// ---- POUs/20_AUTO/Mover/VISU_MoverDetail.TcVIS
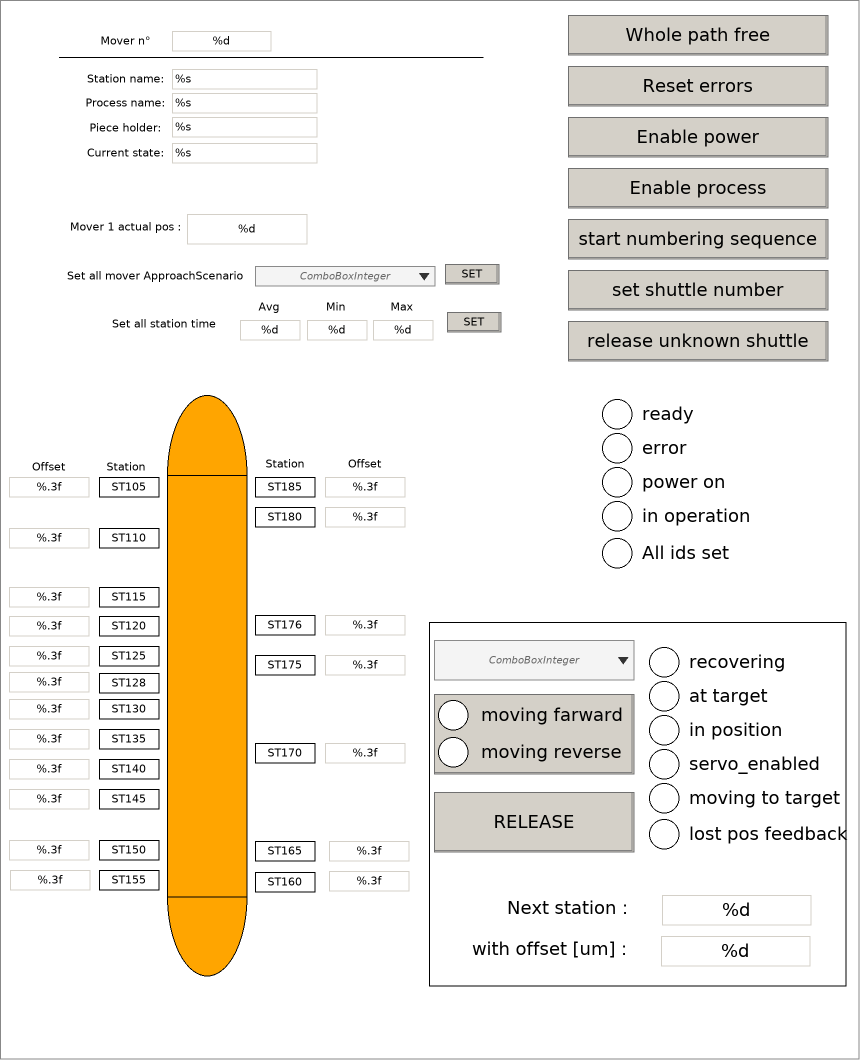
VISUALIZATION VISU_MoverDetail  // 860x1060
    Rectangle (429,622 417x364)
    Button (434,694 200x80)
        toggle gMoverAxis.Q_CT_Shuttle_to_BR.asStruct[HMI.selectedShuttle].bCommand.dirFarward
    Textfield (187,214 120x30), "%d", text variable: MAIN.MoverMan._MoverList[1]._MoverAxis._CurrentPos
        OnMouseDown: write the text variable via Default
    Label (38,212 146x30), "Mover 1 actual pos :"
    ComboBoxInteger (255,266 180x20), variable: MAIN.MoverMan.HMI_Scenario
    Label (59,261 187x30), "Set all mover ApproachScenario"
    Button (445,264 54x20), "SET"
        OnMouseDown: execute { MAIN.MoverMan.SetAllScenario(); }
    Label (93,309 126x30), "Set all station time"
    Textfield (240,320 60x20), "%d", text variable: MAIN.MoverMan.HMI_TimeAvg
        OnMouseDown: write the text variable via Default
    Label (241,296 56x22), "Avg"
    Textfield (307,320 60x20), "%d", text variable: MAIN.MoverMan.HMI_TimeMin
        OnMouseDown: write the text variable via Default
    Label (308,296 56x22), "Min"
    Textfield (373,320 60x20), "%d", text variable: MAIN.MoverMan.HMI_TimeMax
        OnMouseDown: write the text variable via Default
    Label (374,296 56x22), "Max"
    Button (447,312 54x20), "SET"
        OnMouseDown: execute { MAIN.MoverMan.SetAllTimers(ADR(PERS.iStationTimeDef1), 0); MAIN.MoverMan.SetAllTimers(ADR(PERS.iStationTimeDef2), 500); }
    Label (76,26 99x30), "Mover n°"
    Line (59,57) (483,57)
    Label (76,64 99x30), "Station name:"
    Label (76,88 99x30), "Process name:"
    Label (76,113 99x30), "Piece holder:"
    Label (76,138 99x30), "Current state:"
    Textfield (172,31 99x20), "%d", text variable: MAIN.MoverMan.HMI_iSelMover
        OnMouseDown: write the text variable via Default
    Textfield (172,69 145x20), "%s", text variable: MAIN.MoverMan._MoverList[MAIN.MoverMan.HMI_iSelMover].Station.ToString()
    Textfield (172,93 145x20), "%s"
    Textfield (172,117 145x20), "%s", text variable: MAIN.MoverMan._MoverList[MAIN.MoverMan.HMI_iSelMover].AttachedPieceHolder.ToString()
    Textfield (172,143 145x20), "%s", text variable: TO_STRING(MAIN.MoverMan._MoverList[MAIN.MoverMan.HMI_iSelMover]._State)
    Label (79,457 94x20), "Station"
    Label (-1,457 100x20), "Offset"
    Textfield (9,477 80x20), "%.3f", text variable: _20_AUTO.recipe.stationOffsets[StationList_e.ST105]
        OnMouseDown: write the text variable via Default
    Textfield (9,528 80x20), "%.3f", text variable: _20_AUTO.recipe.stationOffsets[StationList_e.ST110]
        OnMouseDown: write the text variable via Default
    Textfield (9,587 80x20), "%.3f", text variable: _20_AUTO.recipe.stationOffsets[StationList_e.ST115]
        OnMouseDown: write the text variable via Default
    Textfield (9,616 80x20), "%.3f", text variable: _20_AUTO.recipe.stationOffsets[StationList_e.ST120]
        OnMouseDown: write the text variable via Default
    Textfield (9,646 80x20), "%.3f", text variable: _20_AUTO.recipe.stationOffsets[StationList_e.ST125]
        OnMouseDown: write the text variable via Default
    Textfield (9,699 80x20), "%.3f", text variable: _20_AUTO.recipe.stationOffsets[StationList_e.ST130]
        OnMouseDown: write the text variable via Default
    Textfield (9,729 80x20), "%.3f", text variable: _20_AUTO.recipe.stationOffsets[StationList_e.ST135]
        OnMouseDown: write the text variable via Default
    Textfield (9,759 80x20), "%.3f", text variable: _20_AUTO.recipe.stationOffsets[StationList_e.ST140]
        OnMouseDown: write the text variable via Default
    Textfield (9,789 80x20), "%.3f", text variable: _20_AUTO.recipe.stationOffsets[StationList_e.ST145]
        OnMouseDown: write the text variable via Default
    Textfield (9,840 80x20), "%.3f", text variable: _20_AUTO.recipe.stationOffsets[StationList_e.ST150]
        OnMouseDown: write the text variable via Default
    Label (315,454 100x20), "Offset"
    Textfield (10,870 80x20), "%.3f", text variable: _20_AUTO.recipe.stationOffsets[StationList_e.ST155]
        OnMouseDown: write the text variable via Default
    Textfield (325,477 80x20), "%.3f", text variable: _20_AUTO.recipe.stationOffsets[StationList_e.ST185]
        OnMouseDown: write the text variable via Default
    Textfield (325,507 80x20), "%.3f", text variable: _20_AUTO.recipe.stationOffsets[StationList_e.ST180]
        OnMouseDown: write the text variable via Default
    Textfield (325,615 80x20), "%.3f", text variable: _20_AUTO.recipe.stationOffsets[StationList_e.ST176]
        OnMouseDown: write the text variable via Default
    Textfield (325,655 80x20), "%.3f", text variable: _20_AUTO.recipe.stationOffsets[StationList_e.ST175]
        OnMouseDown: write the text variable via Default
    Textfield (325,743 80x20), "%.3f", text variable: _20_AUTO.recipe.stationOffsets[StationList_e.ST170]
        OnMouseDown: write the text variable via Default
    Textfield (329,841 80x20), "%.3f", text variable: _20_AUTO.recipe.stationOffsets[StationList_e.ST165]
        OnMouseDown: write the text variable via Default
    Textfield (329,871 80x20), "%.3f", text variable: _20_AUTO.recipe.stationOffsets[StationList_e.ST160]
        OnMouseDown: write the text variable via Default
    Rectangle (99,870 60x20), "ST155", colour toggle: NOT GVL.st155_aut.xMoverPathFree
    Rectangle (99,840 60x20), "ST150", colour toggle: NOT GVL.st150_aut.xMoverPathFree
    Rectangle (99,789 60x20), "ST145", colour toggle: NOT GVL.st145_aut.xMoverPathFree
    Rectangle (99,759 60x20), "ST140", colour toggle: NOT GVL.st140_aut.xMoverPathFree
    Rectangle (99,729 60x20), "ST135", colour toggle: NOT GVL.st135_aut.xMoverPathFree
    Rectangle (99,699 60x20), "ST130", colour toggle: NOT GVL.st130_aut.xMoverPathFree
    Rectangle (99,646 60x20), "ST125", colour toggle: NOT GVL.st125_aut.xMoverPathFree
    Rectangle (99,616 60x20), "ST120", colour toggle: NOT GVL.st120_aut.xMoverPathFree
    Rectangle (99,587 60x20), "ST115", colour toggle: NOT GVL.st115_aut.xMoverPathFree
    Rectangle (99,528 60x20), "ST110", colour toggle: NOT GVL.st110_aut.xMoverPathFree
    Rectangle (99,477 60x20), "ST105", colour toggle: NOT GVL.st105_aut.xMoverPathFree
    Rectangle (255,507 60x20), "ST180", colour toggle: NOT GVL.st180_aut.xMoverPathFree
    Rectangle (255,615 60x20), "ST176", colour toggle: NOT GVL.st176_aut.xMoverPathFree
    Rectangle (255,655 60x20), "ST175", colour toggle: NOT GVL.st175_aut.xMoverPathFree
    Rectangle (255,743 60x20), "ST170", colour toggle: NOT GVL.st170_aut.xMoverPathFree
    Rectangle (255,841 60x20), "ST165", colour toggle: NOT GVL.st165_aut.xMoverPathFree
    Rectangle (255,872 60x20), "ST160", colour toggle: NOT GVL.st160_aut.xMoverPathFree
    Rectangle (255,477 60x20), "ST185", colour toggle: NOT GVL.st185_aut.xMoverPathFree
    Label (238,454 94x20), "Station"
    Ellipse (167,816 80x160)
    Ellipse (167,395 80x160)
    Rectangle (167,475 80x422)
    Button (568,66 260x40), "Reset errors"
        tap gMoverAxis.Q_CT_Track_to_BR.asStruct.bCommand.resetErrors
    Button (568,117 260x40), "Enable power"
        toggle gMoverAxis.Q_CT_Track_to_BR.asStruct.bCommand.enablePower
    ComboBoxInteger (434,640 200x40), variable: HMI.selectedShuttle
    Button (434,792 200x60), "RELEASE", input disabled if: gMoverAxis.Q_CT_Track_to_BR.asStruct.bCommand.enableProcess OR NOT gMoverAxis.I_CT_Track_from_BR.asStruct.bStatus.allIdSet
        tap gMoverAxis.Q_CT_Shuttle_to_BR.asStruct[HMI.selectedShuttle].bCommand.release
    Ellipse (649,647 30x30), colour toggle: gMoverAxis.I_CT_Shuttle_from_BR.asStruct[HMI.selectedShuttle].bStatus.recovering
    Label (686,647 160x30), "recovering"
    Ellipse (649,681 30x30), colour toggle: gMoverAxis.I_CT_Shuttle_from_BR.asStruct[HMI.selectedShuttle].bStatus.at_target
    Label (686,681 160x30), "at target"
    Ellipse (649,715 30x30), colour toggle: gMoverAxis.I_CT_Shuttle_from_BR.asStruct[HMI.selectedShuttle].bStatus.in_position
    Label (686,715 160x30), "in position"
    Ellipse (649,749 30x30), colour toggle: gMoverAxis.I_CT_Shuttle_from_BR.asStruct[HMI.selectedShuttle].bStatus.servo_enabled
    Label (686,749 160x30), "servo_enabled"
    Ellipse (649,783 30x30), colour toggle: gMoverAxis.I_CT_Shuttle_from_BR.asStruct[HMI.selectedShuttle].bStatus.moving_to_load_target
    Label (686,783 160x30), "moving to target"
    Ellipse (649,819 30x30), colour toggle: gMoverAxis.I_CT_Shuttle_from_BR.asStruct[HMI.selectedShuttle].bStatus.lost_position_feedback
    Label (686,819 160x30), "lost pos feedback"
    Ellipse (602,399 30x30), colour toggle: gMoverAxis.I_CT_Track_from_BR.asStruct.bStatus.ready
    Label (639,399 160x30), "ready"
    Ellipse (602,433 30x30), colour toggle: gMoverAxis.I_CT_Track_from_BR.asStruct.bStatus.error
    Label (639,433 160x30), "error"
    Ellipse (602,467 30x30), colour toggle: gMoverAxis.I_CT_Track_from_BR.asStruct.bStatus.powerOn
    Label (639,467 160x30), "power on"
    Ellipse (602,501 30x30), colour toggle: gMoverAxis.I_CT_Track_from_BR.asStruct.bStatus.inOperation
    Label (639,501 160x30), "in operation"
    Button (568,168 260x40), "Enable process"
        toggle gMoverAxis.Q_CT_Track_to_BR.asStruct.bCommand.enableProcess
    Button (568,219 260x40), "start numbering sequence"
        toggle gMoverAxis.Q_CT_Track_to_BR.asStruct.bCommand.startMoverNumberingSequence
    Button (568,270 260x40), "set shuttle number"
        tap gMoverAxis.Q_CT_Track_to_BR.asStruct.bCommand.setShuttleNumber
    Button (568,321 260x40), "release unknown shuttle"
        tap gMoverAxis.Q_CT_Track_to_BR.asStruct.bCommand.releaseUnknownShuttle
    Ellipse (438,700 30x30), colour toggle: gMoverAxis.Q_CT_Shuttle_to_BR.asStruct[HMI.selectedShuttle].bCommand.dirFarward
    Ellipse (438,737 30x30), colour toggle: NOT gMoverAxis.Q_CT_Shuttle_to_BR.asStruct[HMI.selectedShuttle].bCommand.dirFarward
    Label (478,700 160x30), "moving farward"
    Label (478,737 160x30), "moving reverse"
    Button (568,15 260x40), "Whole path free"
        toggle gMoverAxis.Q_CT_Track_to_BR.asStruct.bCommand.wholePathFree
    Textfield (662,895 149x30), "%d", text variable: gMoverAxis.Q_CT_Shuttle_to_BR.asStruct[HMI.selectedShuttle].bNextStation
        OnMouseDown: write the text variable via Default
    Label (471,893 160x30), "Next station :"
    Textfield (661,936 149x30), "%d", text variable: gMoverAxis.Q_CT_Shuttle_to_BR.asStruct[HMI.selectedShuttle].diNextOffset_um
        OnMouseDown: write the text variable via Default
    Label (470,934 160x30), "with offset [um] :"
    Ellipse (602,538 30x30), colour toggle: gMoverAxis.I_CT_Track_from_BR.asStruct.bStatus.allIdSet
    Label (639,538 160x30), "All ids set"
    Textfield (9,672 80x20), "%.3f", text variable: _20_AUTO.recipe.stationOffsets[StationList_e.ST128]
        OnMouseDown: write the text variable via Default
    Rectangle (99,673 60x20), "ST128", colour toggle: NOT GVL.st125_aut.xMoverPathFree
END_VISUALIZATION

// ---- POUs/20_AUTO/Mover/VISU_MoverView.TcVIS
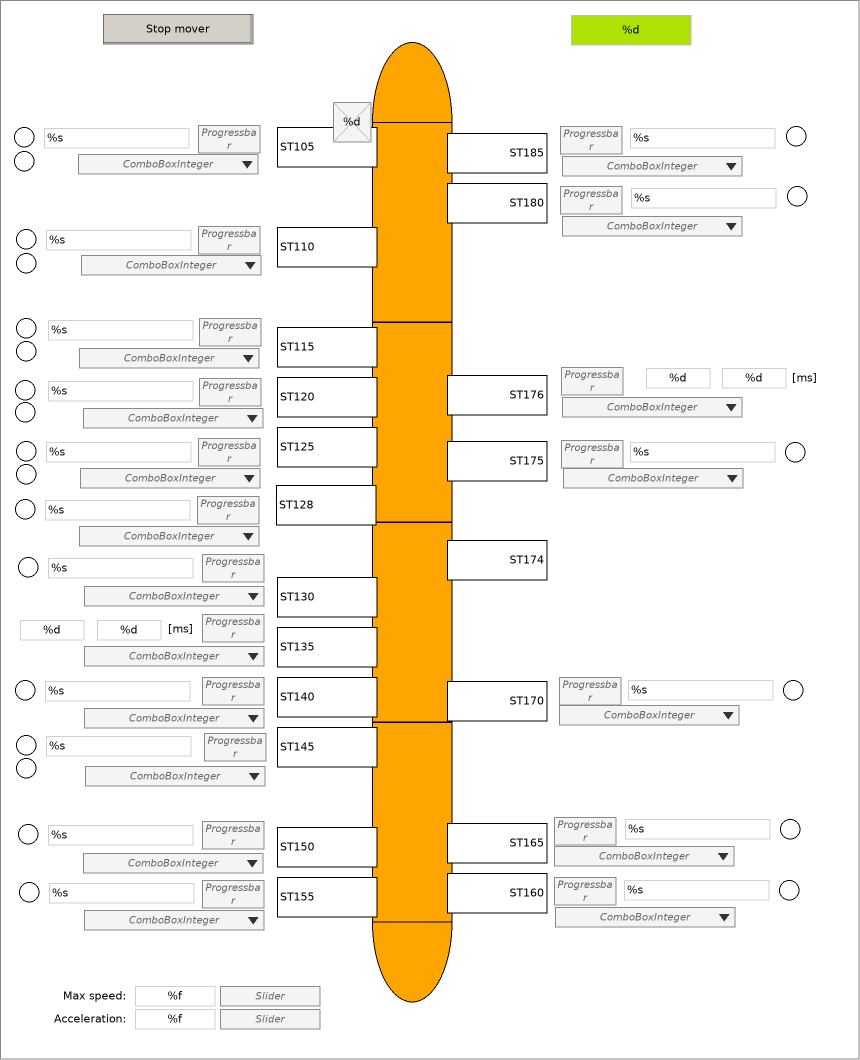
VISUALIZATION VISU_MoverView  // 860x1060
    Ellipse (372,842 80x160)
    Rectangle (372,722 80x200)
    Rectangle (372,522 80x200)
    Rectangle (372,322 80x200)
    Ellipse (372,42 80x160)
    Rectangle (372,122 80x200)
    Rectangle (447,183 100x40), "ST180", colour toggle: NOT GVL.st180_aut.xMoverPathFree
    Rectangle (447,375 100x40), "ST176", colour toggle: NOT GVL.st176_aut.xMoverPathFree
    Rectangle (447,441 100x40), "ST175", colour toggle: NOT GVL.st175_aut.xMoverPathFree
    Rectangle (447,681 100x40), "ST170", colour toggle: NOT GVL.st170_aut.xMoverPathFree
    Rectangle (447,823 100x40), "ST165", colour toggle: NOT GVL.st165_aut.xMoverPathFree
    Rectangle (447,873 100x40), "ST160", colour toggle: NOT GVL.st160_aut.xMoverPathFree
    Rectangle (277,877 100x40), "ST155", colour toggle: NOT GVL.st155_aut.xMoverPathFree
    Rectangle (447,133 100x40), "ST185", colour toggle: NOT GVL.st185_aut.xMoverPathFree
    Progressbar (560,186 62x28), variable: SIMU.iCompletionHMI[18]
    Progressbar (561,367 62x28), variable: SIMU.iCompletionHMI[17]
    Progressbar (561,440 62x28), variable: SIMU.iCompletionHMI[16]
    Progressbar (559,677 62x28), variable: SIMU.iCompletionHMI[14]
    Progressbar (554,817 62x28), variable: SIMU.iCompletionHMI[13]
    Progressbar (554,877 62x28), variable: SIMU.iCompletionHMI[12]
    Progressbar (202,880 62x28), variable: SIMU.iCompletionHMI[11]
    Progressbar (560,126 62x28), variable: SIMU.iCompletionHMI[19]
    Textfield (722,368 64x20), "%d", text variable: PERS.iStationTimeDef2[17]
        OnMouseDown: write the text variable via Default
    Label (777,363 55x30), "[ms]"
    Textfield (571,15 120x30), "%d", text variable: MAIN.MoverMan.PH_num, colour toggle: MAIN.MoverMan.PH_num>2
        OnMouseDown: write the text variable via Default
    ComboBoxInteger (562,156 180x20), variable: MAIN.MoverMan._StationList[18]._ApproachScenario
    ComboBoxInteger (562,216 180x20), variable: MAIN.MoverMan._StationList[17]._ApproachScenario
    ComboBoxInteger (562,397 180x20), variable: MAIN.MoverMan._StationList[16]._ApproachScenario
    ComboBoxInteger (563,468 180x20), variable: MAIN.MoverMan._StationList[16]._ApproachScenario
    ComboBoxInteger (559,705 180x20), variable: MAIN.MoverMan._StationList[14]._ApproachScenario
    ComboBoxInteger (554,846 180x20), variable: MAIN.MoverMan._StationList[13]._ApproachScenario
    ComboBoxInteger (555,907 180x20), variable: MAIN.MoverMan._StationList[12]._ApproachScenario
    ComboBoxInteger (84,910 180x20), variable: MAIN.MoverMan._StationList[11]._ApproachScenario
    Rectangle (277,827 100x40), "ST150", colour toggle: NOT GVL.st150_aut.xMoverPathFree
    Progressbar (202,821 62x28), variable: SIMU.iCompletionHMI[10]
    ComboBoxInteger (83,853 180x20), variable: MAIN.MoverMan._StationList[10]._ApproachScenario
    Rectangle (277,727 100x40), "ST145", colour toggle: NOT GVL.st145_aut.xMoverPathFree
    Progressbar (204,733 62x28), variable: SIMU.iCompletionHMI[9]
    ComboBoxInteger (85,766 180x20), variable: MAIN.MoverMan._StationList[9]._ApproachScenario
    Rectangle (277,677 100x40), "ST140", colour toggle: NOT GVL.st140_aut.xMoverPathFree
    Progressbar (202,677 62x28), variable: SIMU.iCompletionHMI[8]
    ComboBoxInteger (84,708 180x20), variable: MAIN.MoverMan._StationList[8]._ApproachScenario
    Textfield (97,620 64x20), "%d", text variable: PERS.iStationTimeDef2[7]
        OnMouseDown: write the text variable via Default
    Label (153,614 55x30), "[ms]"
    Rectangle (277,627 100x40), "ST135", colour toggle: NOT GVL.st135_aut.xMoverPathFree
    Progressbar (202,614 62x28), variable: SIMU.iCompletionHMI[7]
    ComboBoxInteger (84,646 180x20), variable: MAIN.MoverMan._StationList[7]._ApproachScenario
    Rectangle (277,577 100x40), "ST130", colour toggle: NOT GVL.st130_aut.xMoverPathFree
    Progressbar (202,554 62x28), variable: SIMU.iCompletionHMI[6]
    ComboBoxInteger (84,586 180x20), variable: MAIN.MoverMan._StationList[6]._ApproachScenario
    Rectangle (277,427 100x40), "ST125", colour toggle: NOT GVL.st125_aut.xMoverPathFree
    Progressbar (198,438 62x28), variable: SIMU.iCompletionHMI[5]
    ComboBoxInteger (80,468 180x20), variable: MAIN.MoverMan._StationList[5]._ApproachScenario
    Rectangle (277,377 100x40), "ST120", colour toggle: NOT GVL.st120_aut.xMoverPathFree
    Progressbar (199,378 62x28), variable: SIMU.iCompletionHMI[4]
    ComboBoxInteger (83,408 180x20), variable: MAIN.MoverMan._StationList[4]._ApproachScenario
    Rectangle (277,327 100x40), "ST115", colour toggle: NOT GVL.st115_aut.xMoverPathFree
    Progressbar (199,318 62x28), variable: SIMU.iCompletionHMI[3]
    ComboBoxInteger (79,348 180x20), variable: MAIN.MoverMan._StationList[3]._ApproachScenario
    Rectangle (277,227 100x40), "ST110", colour toggle: NOT GVL.st110_aut.xMoverPathFree
    Progressbar (198,226 62x28), variable: SIMU.iCompletionHMI[2]
    ComboBoxInteger (81,255 180x20), variable: MAIN.MoverMan._StationList[2]._ApproachScenario
    Rectangle (277,127 100x40), "ST105", colour toggle: NOT GVL.st105_aut.xMoverPathFree
    Progressbar (198,125 62x28), variable: SIMU.iCompletionHMI[1]
    ComboBoxInteger (78,154 180x20), variable: MAIN.MoverMan._StationList[1]._ApproachScenario
    Button (103,14 150x30), "Stop mover", colour toggle: MAIN.MoverMan.HMI_xStopMover
        toggle MAIN.MoverMan.HMI_xStopMover
    Textfield (135,986 80x20), "%f", text variable: SIMU.lrSpeedMover
    Textfield (135,1009 80x20), "%f", text variable: SIMU.lrAccelMover
    Label (29,986 100x20), "Max speed:"
    Label (29,1009 100x20), "Acceleration:"
    Slider (220,986 100x20), variable: SIMU.lrSpeedMover, scale 1..50
    Slider (220,1009 100x20), variable: SIMU.lrAccelMoverSlider, scale 0.1..1
    Textfield (20,620 64x20), "%d", text variable: PERS.iStationTimeDef1[7]
        OnMouseDown: write the text variable via Default
    Textfield (646,368 64x20), "%d", text variable: PERS.iStationTimeDef1[17]
        OnMouseDown: write the text variable via Default
    Textfield (46,230 145x20), "%s", text variable: GVL.st110_aut.fb_Pnp.sOUT_Step
    Textfield (48,320 145x20), "%s", text variable: GVL.st115_aut.fb_Pnp.sOUT_Step
    Textfield (48,381 145x20), "%s", text variable: GVL.st120_aut.fb_Pnp.sOUT_Step
    Rectangle (447,540 100x40), "ST174"
    Textfield (46,442 145x20), "%s", text variable: GVL.st125_aut.fb_Pnp.sOUT_Step
    Textfield (46,736 145x20), "%s", text variable: GVL.st145_aut.fb_Pnp.sOUT_Step
    Textfield (631,188 145x20), "%s", text variable: GVL.st180_aut.fb_Pnp.sOUT_Step
    Ellipse (16,229 20x20), colour toggle: GVL.st110_aut.xOUT_Ready
    Ellipse (16,318 20x20), colour toggle: GVL.st115_aut.xOUT_Ready
    Ellipse (15,380 20x20), colour toggle: GVL.st120_aut.xOUT_Ready
    Ellipse (16,441 20x20), colour toggle: GVL.st125_aut.xOUT_Ready
    Ellipse (16,735 20x20), colour toggle: GVL.st145_aut.xOUT_Ready
    Ellipse (787,186 20x20), colour toggle: GVL.st180_aut.xOUT_Ready
    Ellipse (16,253 20x20), colour toggle: GVL.st110_aut.fb_Feeder.xOUT_ErrFlag
    Ellipse (16,341 20x20), colour toggle: GVL.st115_aut.fb_Feeder.xOUT_ErrFlag
    Ellipse (15,402 20x20), colour toggle: GVL.st120_aut.fb_Feeder.xOUT_ErrFlag
    Ellipse (16,464 20x20), colour toggle: GVL.st125_aut.fb_Feeder.xOUT_ErrFlag
    Ellipse (16,758 20x20), colour toggle: GVL.st145_aut.fb_Feeder.xOUT_ErrFlag
    Textfield (630,128 145x20), "%s", text variable: GVL.st185_aut.fb_Pnp.sOUT_Step
    Ellipse (786,126 20x20), colour toggle: GVL.st185_aut.xOUT_Ready
    Textfield (48,558 145x20), "%s", text variable: GVL.st130_aut.fb_Dose.sOUT_Step
    Ellipse (18,557 20x20), colour toggle: GVL.st130_aut.xOUT_Ready
    Textfield (44,128 145x20), "%s", text variable: GVL.st105_aut.fb_Pnp.sOUT_Step
    Ellipse (14,127 20x20), colour toggle: GVL.st105_aut.xOUT_Ready
    Ellipse (14,151 20x20), colour toggle: GVL.st105_aut.fb_Feeder.xOUT_ErrFlag
    Textfield (45,681 145x20), "%s", text variable: GVL.st140_aut.fb_Measure.sOUT_Step
    Ellipse (15,680 20x20), colour toggle: GVL.st140_aut.xOUT_Ready
    Textfield (48,825 145x20), "%s", text variable: GVL.st150_aut.fb_Uss.sOUT_Step
    Ellipse (18,824 20x20), colour toggle: GVL.st150_aut.xOUT_Ready
    Textfield (49,883 145x20), "%s", text variable: GVL.st155_aut.fb_Uss.sOUT_Step
    Ellipse (19,882 20x20), colour toggle: GVL.st155_aut.xOUT_Ready
    Rectangle (276,485 100x40), "ST128", colour toggle: NOT GVL.st128_aut.xMoverPathFree
    Progressbar (197,496 62x28), variable: SIMU.iCompletionHMI[6]
    ComboBoxInteger (79,526 180x20), variable: MAIN.MoverMan._StationList[6]._ApproachScenario
    Textfield (45,500 145x20), "%s", text variable: GVL.st128_aut.fb_TubeCapCheck.sOUT_Step
    Ellipse (15,499 20x20), colour toggle: GVL.st128_aut.xOUT_Ready
    Image (333,102 38x40), "%d", text variable: MAIN.MoverMan._MoverList[1]._ID, colour toggle: MAIN.MoverMan._SimuMoverList[1]._xStuck, invisible if: MAIN.MoverMan._MoverList[1]._MoverAxis._iID>MAIN.MoverMan.MOVER_NUMBER, image: Custom.MoverSimu_final
        p3560616238: MAIN.MoverMan._MoverList[1]._MoverAxis.outSimuCurrentPos.x
        p2738717112: MAIN.MoverMan._MoverList[1]._MoverAxis.outSimuCurrentPos.y
        p2858320360: -MAIN.MoverMan._MoverList[1]._MoverAxis.outSimuCurrentRot
    Image (333,102 38x40), "%d", text variable: MAIN.MoverMan._MoverList[2]._ID, colour toggle: MAIN.MoverMan._SimuMoverList[2]._xStuck, invisible if: MAIN.MoverMan._MoverList[2]._MoverAxis._iID>MAIN.MoverMan.MOVER_NUMBER, image: Custom.MoverSimu_final
        p3560616238: MAIN.MoverMan._MoverList[2]._MoverAxis.outSimuCurrentPos.x
        p2738717112: MAIN.MoverMan._MoverList[2]._MoverAxis.outSimuCurrentPos.y
        p2858320360: -MAIN.MoverMan._MoverList[2]._MoverAxis.outSimuCurrentRot
    Image (333,102 38x40), "%d", text variable: MAIN.MoverMan._MoverList[3]._ID, colour toggle: MAIN.MoverMan._SimuMoverList[3]._xStuck, invisible if: MAIN.MoverMan._MoverList[3]._MoverAxis._iID>MAIN.MoverMan.MOVER_NUMBER, image: Custom.MoverSimu_final
        p3560616238: MAIN.MoverMan._MoverList[3]._MoverAxis.outSimuCurrentPos.x
        p2738717112: MAIN.MoverMan._MoverList[3]._MoverAxis.outSimuCurrentPos.y
        p2858320360: -MAIN.MoverMan._MoverList[3]._MoverAxis.outSimuCurrentRot
    Image (333,102 38x40), "%d", text variable: MAIN.MoverMan._MoverList[4]._ID, colour toggle: MAIN.MoverMan._SimuMoverList[4]._xStuck, invisible if: MAIN.MoverMan._MoverList[4]._MoverAxis._iID>MAIN.MoverMan.MOVER_NUMBER, image: Custom.MoverSimu_final
        p3560616238: MAIN.MoverMan._MoverList[4]._MoverAxis.outSimuCurrentPos.x
        p2738717112: MAIN.MoverMan._MoverList[4]._MoverAxis.outSimuCurrentPos.y
        p2858320360: -MAIN.MoverMan._MoverList[4]._MoverAxis.outSimuCurrentRot
    Image (333,102 38x40), "%d", text variable: MAIN.MoverMan._MoverList[5]._ID, colour toggle: MAIN.MoverMan._SimuMoverList[5]._xStuck, invisible if: MAIN.MoverMan._MoverList[5]._MoverAxis._iID>MAIN.MoverMan.MOVER_NUMBER, image: Custom.MoverSimu_final
        p3560616238: MAIN.MoverMan._MoverList[5]._MoverAxis.outSimuCurrentPos.x
        p2738717112: MAIN.MoverMan._MoverList[5]._MoverAxis.outSimuCurrentPos.y
        p2858320360: -MAIN.MoverMan._MoverList[5]._MoverAxis.outSimuCurrentRot
    Image (333,102 38x40), "%d", text variable: MAIN.MoverMan._MoverList[6]._ID, colour toggle: MAIN.MoverMan._SimuMoverList[6]._xStuck, invisible if: MAIN.MoverMan._MoverList[6]._MoverAxis._iID>MAIN.MoverMan.MOVER_NUMBER, image: Custom.MoverSimu_final
        p3560616238: MAIN.MoverMan._MoverList[6]._MoverAxis.outSimuCurrentPos.x
        p2738717112: MAIN.MoverMan._MoverList[6]._MoverAxis.outSimuCurrentPos.y
        p2858320360: -MAIN.MoverMan._MoverList[6]._MoverAxis.outSimuCurrentRot
    Image (333,102 38x40), "%d", text variable: MAIN.MoverMan._MoverList[7]._ID, colour toggle: MAIN.MoverMan._SimuMoverList[7]._xStuck, invisible if: MAIN.MoverMan._MoverList[7]._MoverAxis._iID>MAIN.MoverMan.MOVER_NUMBER, image: Custom.MoverSimu_final
        p3560616238: MAIN.MoverMan._MoverList[7]._MoverAxis.outSimuCurrentPos.x
        p2738717112: MAIN.MoverMan._MoverList[7]._MoverAxis.outSimuCurrentPos.y
        p2858320360: -MAIN.MoverMan._MoverList[7]._MoverAxis.outSimuCurrentRot
    Image (333,102 38x40), "%d", text variable: MAIN.MoverMan._MoverList[8]._ID, colour toggle: MAIN.MoverMan._SimuMoverList[8]._xStuck, invisible if: MAIN.MoverMan._MoverList[8]._MoverAxis._iID>MAIN.MoverMan.MOVER_NUMBER, image: Custom.MoverSimu_final
        p3560616238: MAIN.MoverMan._MoverList[8]._MoverAxis.outSimuCurrentPos.x
        p2738717112: MAIN.MoverMan._MoverList[8]._MoverAxis.outSimuCurrentPos.y
        p2858320360: -MAIN.MoverMan._MoverList[8]._MoverAxis.outSimuCurrentRot
    Image (333,102 38x40), "%d", text variable: MAIN.MoverMan._MoverList[9]._ID, colour toggle: MAIN.MoverMan._SimuMoverList[9]._xStuck, invisible if: MAIN.MoverMan._MoverList[9]._MoverAxis._iID>MAIN.MoverMan.MOVER_NUMBER, image: Custom.MoverSimu_final
        p3560616238: MAIN.MoverMan._MoverList[9]._MoverAxis.outSimuCurrentPos.x
        p2738717112: MAIN.MoverMan._MoverList[9]._MoverAxis.outSimuCurrentPos.y
        p2858320360: -MAIN.MoverMan._MoverList[9]._MoverAxis.outSimuCurrentRot
    Image (333,102 38x40), "%d", text variable: MAIN.MoverMan._MoverList[10]._ID, colour toggle: MAIN.MoverMan._SimuMoverList[10]._xStuck, invisible if: MAIN.MoverMan._MoverList[10]._MoverAxis._iID>MAIN.MoverMan.MOVER_NUMBER, image: Custom.MoverSimu_final
        p3560616238: MAIN.MoverMan._MoverList[10]._MoverAxis.outSimuCurrentPos.x
        p2738717112: MAIN.MoverMan._MoverList[10]._MoverAxis.outSimuCurrentPos.y
        p2858320360: -MAIN.MoverMan._MoverList[10]._MoverAxis.outSimuCurrentRot
    Image (333,102 38x40), "%d", text variable: MAIN.MoverMan._MoverList[11]._ID, colour toggle: MAIN.MoverMan._SimuMoverList[11]._xStuck, invisible if: MAIN.MoverMan._MoverList[11]._MoverAxis._iID>MAIN.MoverMan.MOVER_NUMBER, image: Custom.MoverSimu_final
        p3560616238: MAIN.MoverMan._MoverList[11]._MoverAxis.outSimuCurrentPos.x
        p2738717112: MAIN.MoverMan._MoverList[11]._MoverAxis.outSimuCurrentPos.y
        p2858320360: -MAIN.MoverMan._MoverList[11]._MoverAxis.outSimuCurrentRot
    Image (333,102 38x40), "%d", text variable: MAIN.MoverMan._MoverList[12]._ID, colour toggle: MAIN.MoverMan._SimuMoverList[12]._xStuck, invisible if: MAIN.MoverMan._MoverList[12]._MoverAxis._iID>MAIN.MoverMan.MOVER_NUMBER, image: Custom.MoverSimu_final
        p3560616238: MAIN.MoverMan._MoverList[12]._MoverAxis.outSimuCurrentPos.x
        p2738717112: MAIN.MoverMan._MoverList[12]._MoverAxis.outSimuCurrentPos.y
        p2858320360: -MAIN.MoverMan._MoverList[12]._MoverAxis.outSimuCurrentRot
    Image (333,102 38x40), "%d", text variable: MAIN.MoverMan._MoverList[13]._ID, colour toggle: MAIN.MoverMan._SimuMoverList[13]._xStuck, invisible if: MAIN.MoverMan._MoverList[13]._MoverAxis._iID>MAIN.MoverMan.MOVER_NUMBER, image: Custom.MoverSimu_final
        p3560616238: MAIN.MoverMan._MoverList[13]._MoverAxis.outSimuCurrentPos.x
        p2738717112: MAIN.MoverMan._MoverList[13]._MoverAxis.outSimuCurrentPos.y
        p2858320360: -MAIN.MoverMan._MoverList[13]._MoverAxis.outSimuCurrentRot
    Image (333,102 38x40), "%d", text variable: MAIN.MoverMan._MoverList[14]._ID, colour toggle: MAIN.MoverMan._SimuMoverList[14]._xStuck, invisible if: MAIN.MoverMan._MoverList[14]._MoverAxis._iID>MAIN.MoverMan.MOVER_NUMBER, image: Custom.MoverSimu_final
        p3560616238: MAIN.MoverMan._MoverList[14]._MoverAxis.outSimuCurrentPos.x
        p2738717112: MAIN.MoverMan._MoverList[14]._MoverAxis.outSimuCurrentPos.y
        p2858320360: -MAIN.MoverMan._MoverList[14]._MoverAxis.outSimuCurrentRot
    Image (333,102 38x40), "%d", text variable: MAIN.MoverMan._MoverList[15]._ID, colour toggle: MAIN.MoverMan._SimuMoverList[15]._xStuck, invisible if: MAIN.MoverMan._MoverList[15]._MoverAxis._iID>MAIN.MoverMan.MOVER_NUMBER, image: Custom.MoverSimu_final
        p3560616238: MAIN.MoverMan._MoverList[15]._MoverAxis.outSimuCurrentPos.x
        p2738717112: MAIN.MoverMan._MoverList[15]._MoverAxis.outSimuCurrentPos.y
        p2858320360: -MAIN.MoverMan._MoverList[15]._MoverAxis.outSimuCurrentRot
    Image (333,102 38x40), "%d", text variable: MAIN.MoverMan._MoverList[16]._ID, colour toggle: MAIN.MoverMan._SimuMoverList[16]._xStuck, invisible if: MAIN.MoverMan._MoverList[16]._MoverAxis._iID>MAIN.MoverMan.MOVER_NUMBER, image: Custom.MoverSimu_final
        p3560616238: MAIN.MoverMan._MoverList[16]._MoverAxis.outSimuCurrentPos.x
        p2738717112: MAIN.MoverMan._MoverList[16]._MoverAxis.outSimuCurrentPos.y
        p2858320360: -MAIN.MoverMan._MoverList[16]._MoverAxis.outSimuCurrentRot
    Image (333,102 38x40), "%d", text variable: MAIN.MoverMan._MoverList[17]._ID, colour toggle: MAIN.MoverMan._SimuMoverList[17]._xStuck, invisible if: MAIN.MoverMan._MoverList[17]._MoverAxis._iID>MAIN.MoverMan.MOVER_NUMBER, image: Custom.MoverSimu_final
        p3560616238: MAIN.MoverMan._MoverList[17]._MoverAxis.outSimuCurrentPos.x
        p2738717112: MAIN.MoverMan._MoverList[17]._MoverAxis.outSimuCurrentPos.y
        p2858320360: -MAIN.MoverMan._MoverList[17]._MoverAxis.outSimuCurrentRot
    Image (333,102 38x40), "%d", text variable: MAIN.MoverMan._MoverList[18]._ID, colour toggle: MAIN.MoverMan._SimuMoverList[18]._xStuck, invisible if: MAIN.MoverMan._MoverList[18]._MoverAxis._iID>MAIN.MoverMan.MOVER_NUMBER, image: Custom.MoverSimu_final
        p3560616238: MAIN.MoverMan._MoverList[18]._MoverAxis.outSimuCurrentPos.x
        p2738717112: MAIN.MoverMan._MoverList[18]._MoverAxis.outSimuCurrentPos.y
        p2858320360: -MAIN.MoverMan._MoverList[18]._MoverAxis.outSimuCurrentRot
    Image (333,102 38x40), "%d", text variable: MAIN.MoverMan._MoverList[19]._ID, colour toggle: MAIN.MoverMan._SimuMoverList[19]._xStuck, invisible if: MAIN.MoverMan._MoverList[19]._MoverAxis._iID>MAIN.MoverMan.MOVER_NUMBER, image: Custom.MoverSimu_final
        p3560616238: MAIN.MoverMan._MoverList[19]._MoverAxis.outSimuCurrentPos.x
        p2738717112: MAIN.MoverMan._MoverList[19]._MoverAxis.outSimuCurrentPos.y
        p2858320360: -MAIN.MoverMan._MoverList[19]._MoverAxis.outSimuCurrentRot
    Textfield (624,880 145x20), "%s", text variable: GVL.st160_aut.fb_ABL_CETA.sOUT_Step
    Ellipse (779,880 20x20), colour toggle: GVL.st160_aut.xOUT_Ready
    Textfield (625,819 145x20), "%s", text variable: GVL.st165_aut.fb_ABL_CETA.sOUT_Step
    Ellipse (780,819 20x20), colour toggle: GVL.st160_aut.xOUT_Ready
    Textfield (628,680 145x20), "%s", text variable: GVL.st170_aut.fb_ABL_RFID.sOUT_Step
    Ellipse (783,680 20x20), colour toggle: GVL.st170_aut.xOUT_Ready
    Textfield (630,442 145x20), "%s", text variable: GVL.st175_aut.fb_laser.sOUT_Step
    Ellipse (785,442 20x20), colour toggle: GVL.st175_aut.xOUT_Ready
END_VISUALIZATION

// ---- POUs/20_AUTO/ST105/VISU_Recipe_ST105.TcVIS
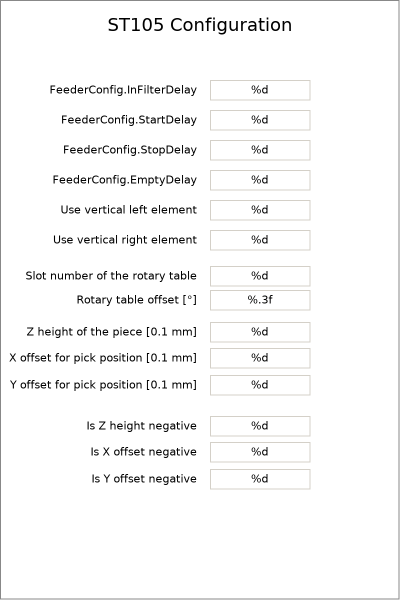
VISUALIZATION VISU_Recipe_ST105  // 400x600
    Textfield (210,80 100x20), "%d", text variable: _20_AUTO.recipe.st110.FeederConfig.InFilterDelay
        OnMouseDown: write the text variable via Default
    Label (0,5 400x40), "ST105 Configuration"
    Label (0,80 200x20), "FeederConfig.InFilterDelay"
    Textfield (210,110 100x20), "%d", text variable: _20_AUTO.recipe.st110.FeederConfig.StartDelay
        OnMouseDown: write the text variable via Default
    Label (0,110 200x20), "FeederConfig.StartDelay"
    Textfield (210,140 100x20), "%d", text variable: _20_AUTO.recipe.st105.FeederConfig.StopDelay
        OnMouseDown: write the text variable via Default
    Label (0,140 200x20), "FeederConfig.StopDelay"
    Textfield (210,170 100x20), "%d", text variable: _20_AUTO.recipe.st105.FeederConfig.EmptyDelay
        OnMouseDown: write the text variable via Default
    Label (0,170 200x20), "FeederConfig.EmptyDelay"
    Label (0,200 200x20), "Use vertical left element"
    Label (0,230 200x20), "Use vertical right element"
    Textfield (210,200 100x20), "%d", text variable: _20_AUTO.recipe.st105.xUseVerLeft
        OnMouseDown: write the text variable via Default
    Textfield (210,230 100x20), "%d", text variable: _20_AUTO.recipe.st105.xUseVerRight
        OnMouseDown: write the text variable via Default
    Textfield (210,416 100x20), "%d", text variable: _20_AUTO.recipe.st105.isPickUpPos_Z_neg
        OnMouseDown: write the text variable via Default
    Label (0,442 200x20), "Is X offset negative"
    Textfield (210,442 100x20), "%d", text variable: _20_AUTO.recipe.st105.isPickOffset_X_neg
        OnMouseDown: write the text variable via Default
    Label (0,469 200x20), "Is Y offset negative"
    Textfield (210,469 100x20), "%d", text variable: _20_AUTO.recipe.st105.isPickOffset_Y_neg
        OnMouseDown: write the text variable via Default
    Label (0,416 200x20), "Is Z height negative"
    Textfield (210,322 100x20), "%d", text variable: _20_AUTO.recipe.st105.PickUpPos_Z_deci
        OnMouseDown: write the text variable via Default
    Label (0,348 200x20), "X offset for pick position [0.1 mm]"
    Textfield (210,348 100x20), "%d", text variable: _20_AUTO.recipe.st105.PickOffset_X_deci
        OnMouseDown: write the text variable via Default
    Label (0,375 200x20), "Y offset for pick position [0.1 mm]"
    Textfield (210,375 100x20), "%d", text variable: _20_AUTO.recipe.st105.PickOffset_Y_deci
        OnMouseDown: write the text variable via Default
    Label (0,322 200x20), "Z height of the piece [0.1 mm]"
    Label (0,266 200x20), "Slot number of the rotary table"
    Textfield (210,266 100x20), "%d", text variable: _20_AUTO.recipe.st105.FeederSize
        OnMouseDown: write the text variable via Default
    Textfield (210,290 100x20), "%.3f", text variable: _20_AUTO.recipe.st105.RotaryTableOffset
        OnMouseDown: write the text variable via Default
    Label (0,290 200x20), "Rotary table offset [°]"
END_VISUALIZATION

// ---- POUs/20_AUTO/ST105/VISU_ST105.TcVIS
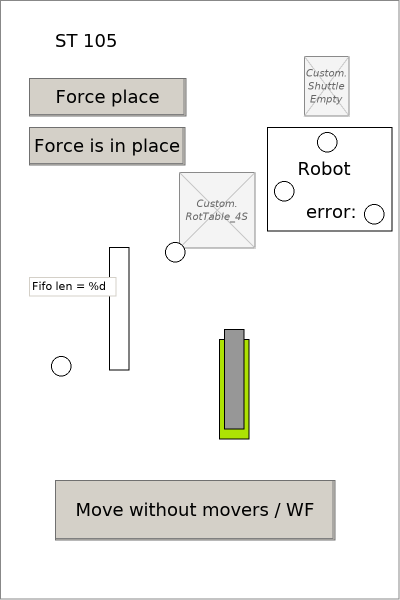
VISUALIZATION VISU_ST105  // 400x600
    Image (304,56 45x60), angle 90, invisible if: NOT __ISVALIDREF(GVL.st105_aut._Mover), image: Custom.Shuttle Empty
    Image (179,172 76x76), angle 45, image: Custom.RotTable_4S
        p2858320360: ST105_Axis.axis105_10W.rActPos
    Rectangle (109,247 20x123), angle 45
    Ellipse (51,356 20x20), colour toggle: GVL.st105_aut.fb_Feeder.simu_feeder.xOUT_NewPiece
    Ellipse (165,242 20x20), colour toggle: GVL.st105_aut.fb_Feeder.simu_feeder.xOUT_NewPiece
    Textfield (29,277 87x19), "Fifo len = %d", text variable: GVL.st105_aut.fb_Feeder.simu_fifo_feeder_to_rotTable.GetLen()
    Label (44,31 85x20), "ST 105"
    Rectangle (219,339 30x100)
    Rectangle (224,329 20x100)
        p2738717112: -GVL.st105_aut.fb_Pnp.fb_simu_axis105_11Z.rOUT_PixActual
    Button (55,480 280x60), "Move without movers / WF", colour toggle: HMI.bArForceCyclusState[StationList_e.ST105]
        tap HMI.btArForceCyclus[StationList_e.ST105].button
    Rectangle (267,127 125x104)
    Ellipse (274,181 20x20), colour toggle: GVL.st105_aut.fb_Pnp.aut_status_from_robot.Picked
    Ellipse (317,132 20x20), colour toggle: GVL.st105_aut.fb_Pnp.aut_status_from_robot.Placed
    Ellipse (364,204 20x20), colour toggle: GVL.st105_aut.fb_Pnp.fanuc_status.Fault
    Label (283,154 82x30), "Robot"
    Label (299,197 65x30), "error:"
    Button (29,78 157x38), "Force place", colour toggle: HMI.bArForceCyclusState[StationList_e.ST105]
        tap GVL.st105_aut.fb_Pnp.hmi_force_place
    Button (29,127 156x38), "Force is in place", colour toggle: HMI.bArForceCyclusState[StationList_e.ST105]
        tap GVL.st105_aut.fb_Pnp.hmi_force_in_place
END_VISUALIZATION

// ---- POUs/20_AUTO/ST110/VISU_Recipe_ST110.TcVIS
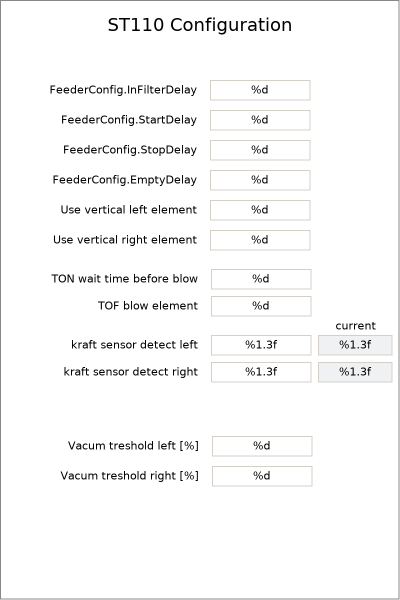
VISUALIZATION VISU_Recipe_ST110  // 400x600
    Textfield (210,80 100x20), "%d", text variable: _20_AUTO.recipe.st110.FeederConfig.InFilterDelay
        OnMouseDown: write the text variable via Default
    Label (0,5 400x40), "ST110 Configuration"
    Label (0,80 200x20), "FeederConfig.InFilterDelay"
    Textfield (210,110 100x20), "%d", text variable: _20_AUTO.recipe.st110.FeederConfig.StartDelay
        OnMouseDown: write the text variable via Default
    Label (0,110 200x20), "FeederConfig.StartDelay"
    Textfield (210,140 100x20), "%d", text variable: _20_AUTO.recipe.st110.FeederConfig.StopDelay
        OnMouseDown: write the text variable via Default
    Label (0,140 200x20), "FeederConfig.StopDelay"
    Textfield (210,170 100x20), "%d", text variable: _20_AUTO.recipe.st110.FeederConfig.EmptyDelay
        OnMouseDown: write the text variable via Default
    Label (0,170 200x20), "FeederConfig.EmptyDelay"
    Label (0,200 200x20), "Use vertical left element"
    Label (0,230 200x20), "Use vertical right element"
    Textfield (210,200 100x20), "%d", text variable: _20_AUTO.recipe.st110.xUseVerLeft
        OnMouseDown: write the text variable via Default
    Textfield (210,230 100x20), "%d", text variable: _20_AUTO.recipe.st110.xUseVerRight
        OnMouseDown: write the text variable via Default
    Label (1,296 200x20), "TOF blow element"
    Textfield (211,296 100x20), "%d", text variable: _20_AUTO.recipe.st110.blowPieceTof_ms
        OnMouseDown: write the text variable via Default
    Label (2,436 200x20), "Vacum treshold left [%]"
    Label (2,466 200x20), "Vacum treshold right [%]"
    Textfield (212,436 100x20), "%d", text variable: _20_AUTO.recipe.st110.vakum_left_pc
        OnMouseDown: write the text variable via Default
    Textfield (212,466 100x20), "%d", text variable: _20_AUTO.recipe.st110.vakum_right_pc
        OnMouseDown: write the text variable via Default
    Label (1,269 200x20), "TON wait time before blow"
    Textfield (211,269 100x20), "%d", text variable: _20_AUTO.recipe.st110.waitBlowPieceTon_ms
        OnMouseDown: write the text variable via Default
    Label (1,362 200x20), "kraft sensor detect right"
    Textfield (211,362 100x20), "%1.3f", text variable: _20_AUTO.recipe.st110.kraft_right_raw
        OnMouseDown: write the text variable via Default
    Label (1,335 200x20), "kraft sensor detect left"
    Textfield (211,335 100x20), "%1.3f", text variable: _20_AUTO.recipe.st110.kraft_left_raw
        OnMouseDown: write the text variable via Default
    Textfield (318,335 74x20), "%1.3f", text variable: GVL.st110_aut.fb_Pnp.fb_kraftLeft.lrOUT_value
        OnMouseDown: write the text variable via Default
    Textfield (318,362 74x20), "%1.3f", text variable: GVL.st110_aut.fb_Pnp.fb_kraftRight.lrOUT_value
        OnMouseDown: write the text variable via Default
    Label (321,316 70x20), "current"
END_VISUALIZATION

// ---- POUs/20_AUTO/ST110/VISU_ST110.TcVIS
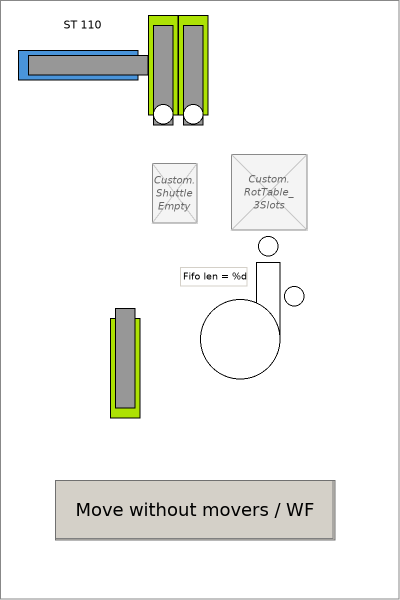
VISUALIZATION VISU_ST110  // 400x600
    Image (152,163 45x60), invisible if: NOT __ISVALIDREF(GVL.st110_aut._Mover), image: Custom.Shuttle Empty
    Image (231,154 76x76), image: Custom.RotTable_3Slots
        p2858320360: ST110_Axis.axis110_10W.rActPos
    Rectangle (18,50 120x30)
    Rectangle (28,55 120x20)
        p3560616238: GVL.st110_aut.fb_Pnp.fb_simu_axis110_01Y.rOUT_PixActual
    Rectangle (148,15 30x100)
        p3560616238: GVL.st110_aut.fb_Pnp.fb_simu_axis110_01Y.rOUT_PixActual
    Rectangle (153,25 20x100)
        p2738717112: GVL.st110_aut.fb_Pnp.fb_simu_axis110_02Z.rOUT_PixActual
        p3560616238: GVL.st110_aut.fb_Pnp.fb_simu_axis110_01Y.rOUT_PixActual
    Rectangle (178,15 30x100)
        p3560616238: GVL.st110_aut.fb_Pnp.fb_simu_axis110_01Y.rOUT_PixActual
    Rectangle (183,25 20x100)
        p2738717112: GVL.st110_aut.fb_Pnp.fb_simu_axis110_03Z.rOUT_PixActual
        p3560616238: GVL.st110_aut.fb_Pnp.fb_simu_axis110_01Y.rOUT_PixActual
    Rectangle (256,262 24x73)
    Ellipse (200,299 80x80), colour toggle: GVL.st110_aut.fb_Feeder.simu_feeder.xIN_Enable
    Ellipse (284,286 20x20), colour toggle: GVL.st110_aut.fb_Feeder.simu_feeder.xOUT_NewPiece
    Ellipse (153,104 20x20), colour toggle: GVL.st110_aut.fb_Pnp.fb_gripperLeft.xIN_AS
        p3560616238: GVL.st110_aut.fb_Pnp.fb_simu_axis110_01Y.rOUT_PixActual
        p2738717112: GVL.st110_aut.fb_Pnp.fb_simu_axis110_02Z.rOUT_PixActual
    Ellipse (183,104 20x20), colour toggle: GVL.st110_aut.fb_Pnp.fb_gripperRight.xIN_AS
        p2738717112: GVL.st110_aut.fb_Pnp.fb_simu_axis110_03Z.rOUT_PixActual
        p3560616238: GVL.st110_aut.fb_Pnp.fb_simu_axis110_01Y.rOUT_PixActual
    Ellipse (258,236 20x20), colour toggle: GVL.st110_aut.fb_Feeder.simu_feeder.xOUT_NewPiece
    Textfield (180,267 67x19), "Fifo len = %d", text variable: GVL.st110_aut.fb_Feeder.simu_fifo_feeder_to_rotTable.GetLen()
    Label (40,15 85x20), "ST 110"
    Rectangle (110,318 30x100)
    Rectangle (115,308 20x100)
        p2738717112: -GVL.st110_aut.fb_Pnp.fb_simu_axis110_04Z.rOUT_PixActual
    Button (55,480 280x60), "Move without movers / WF", colour toggle: HMI.bArForceCyclusState[StationList_e.ST110]
        tap HMI.btArForceCyclus[StationList_e.ST110].button
END_VISUALIZATION

// ---- POUs/20_AUTO/ST115/VISU_Recipe_ST115.TcVIS
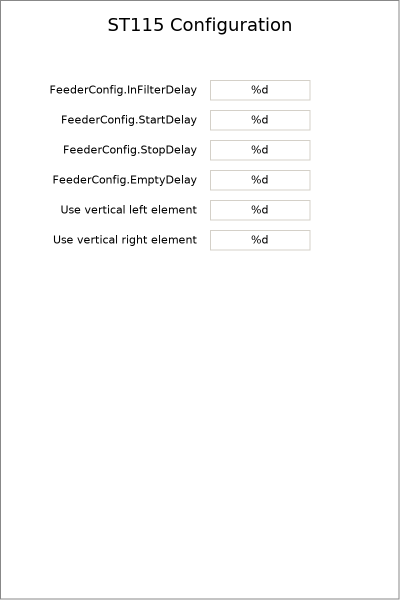
VISUALIZATION VISU_Recipe_ST115  // 400x600
    Textfield (210,80 100x20), "%d", text variable: _20_AUTO.recipe.st115.FeederConfig.InFilterDelay
        OnMouseDown: write the text variable via Default
    Label (0,5 400x40), "ST115 Configuration"
    Label (0,80 200x20), "FeederConfig.InFilterDelay"
    Textfield (210,110 100x20), "%d", text variable: _20_AUTO.recipe.st115.FeederConfig.StartDelay
        OnMouseDown: write the text variable via Default
    Label (0,110 200x20), "FeederConfig.StartDelay"
    Textfield (210,140 100x20), "%d", text variable: _20_AUTO.recipe.st115.FeederConfig.StopDelay
        OnMouseDown: write the text variable via Default
    Label (0,140 200x20), "FeederConfig.StopDelay"
    Textfield (210,170 100x20), "%d", text variable: _20_AUTO.recipe.st115.FeederConfig.EmptyDelay
        OnMouseDown: write the text variable via Default
    Label (0,170 200x20), "FeederConfig.EmptyDelay"
    Label (0,200 200x20), "Use vertical left element"
    Label (0,230 200x20), "Use vertical right element"
    Textfield (210,200 100x20), "%d", text variable: _20_AUTO.recipe.st115.xUseVerLeft
        OnMouseDown: write the text variable via Default
    Textfield (210,230 100x20), "%d", text variable: _20_AUTO.recipe.st115.xUseVerRight
        OnMouseDown: write the text variable via Default
END_VISUALIZATION

// ---- POUs/20_AUTO/ST115/VISU_ST115.TcVIS
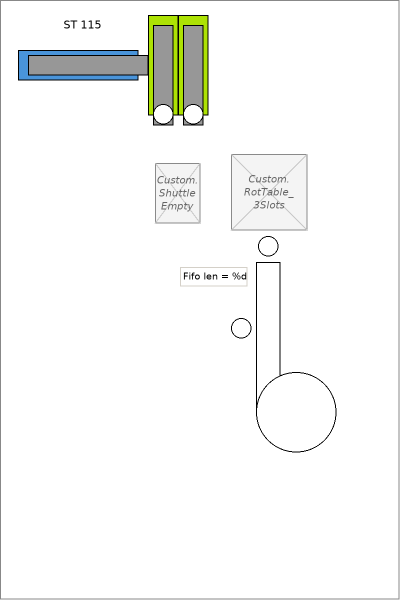
VISUALIZATION VISU_ST115  // 400x600
    Image (155,163 45x60), invisible if: NOT __ISVALIDREF(GVL.st115_aut._Mover), image: Custom.Shuttle Empty
    Image (231,154 76x76), image: Custom.RotTable_3Slots
        p2858320360: ST115_Axis.axis115_10W.rActPos
    Rectangle (18,50 120x30)
    Rectangle (28,55 120x20)
        p3560616238: GVL.st115_aut.fb_Pnp.fb_simu_axis115_01Y.rOUT_PixActual
    Rectangle (148,15 30x100)
        p3560616238: GVL.st115_aut.fb_Pnp.fb_simu_axis115_01Y.rOUT_PixActual
    Rectangle (153,25 20x100)
        p2738717112: GVL.st115_aut.fb_Pnp.fb_simu_axis115_02Z.rOUT_PixActual
        p3560616238: GVL.st115_aut.fb_Pnp.fb_simu_axis115_01Y.rOUT_PixActual
    Rectangle (178,15 30x100)
        p3560616238: GVL.st115_aut.fb_Pnp.fb_simu_axis115_01Y.rOUT_PixActual
    Rectangle (183,25 20x100)
        p2738717112: GVL.st115_aut.fb_Pnp.fb_simu_axis115_03Z.rOUT_PixActual
        p3560616238: GVL.st115_aut.fb_Pnp.fb_simu_axis115_01Y.rOUT_PixActual
    Rectangle (256,262 24x150)
    Ellipse (256,372 80x80), colour toggle: GVL.st115_aut.fb_Feeder.simu_feeder.xIN_Enable
    Ellipse (231,318 20x20), colour toggle: GVL.st115_aut.fb_Feeder.simu_feeder.xOUT_NewPiece
    Ellipse (153,104 20x20), colour toggle: GVL.st115_aut.fb_Pnp.fb_gripperLeft.xIN_AS
        p3560616238: GVL.st115_aut.fb_Pnp.fb_simu_axis115_01Y.rOUT_PixActual
        p2738717112: GVL.st115_aut.fb_Pnp.fb_simu_axis115_02Z.rOUT_PixActual
    Ellipse (183,104 20x20), colour toggle: GVL.st115_aut.fb_Pnp.fb_gripperRight.xIN_AS
        p2738717112: GVL.st115_aut.fb_Pnp.fb_simu_axis115_02Z.rOUT_PixActual
        p3560616238: GVL.st115_aut.fb_Pnp.fb_simu_axis115_01Y.rOUT_PixActual
    Ellipse (258,236 20x20), colour toggle: NOT GVL.st115_aut.fb_Feeder.simu_feeder.xOUT_NewPiece
    Textfield (180,267 67x19), "Fifo len = %d", text variable: GVL.st115_aut.fb_Feeder.simu_fifo_feeder_to_rotTable.GetLen()
    Label (40,15 85x20), "ST 115"
END_VISUALIZATION

// ---- POUs/20_AUTO/ST120/VISU_Recipe_ST120.TcVIS
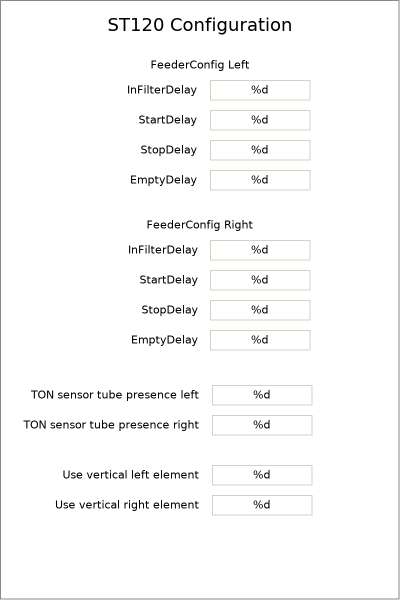
VISUALIZATION VISU_Recipe_ST120  // 400x600
    Textfield (210,80 100x20), "%d", text variable: _20_AUTO.recipe.st120.FeederConfigLeft.InFilterDelay
        OnMouseDown: write the text variable via Default
    Label (0,5 400x40), "ST120 Configuration"
    Label (0,80 200x20), "InFilterDelay"
    Textfield (210,110 100x20), "%d", text variable: _20_AUTO.recipe.st120.FeederConfigLeft.StartDelay
        OnMouseDown: write the text variable via Default
    Label (0,110 200x20), "StartDelay"
    Textfield (210,140 100x20), "%d", text variable: _20_AUTO.recipe.st120.FeederConfigLeft.StopDelay
        OnMouseDown: write the text variable via Default
    Label (0,140 200x20), "StopDelay"
    Textfield (210,170 100x20), "%d", text variable: _20_AUTO.recipe.st120.FeederConfigLeft.EmptyDelay
        OnMouseDown: write the text variable via Default
    Label (0,170 200x20), "EmptyDelay"
    Label (2,465 200x20), "Use vertical left element"
    Label (2,495 200x20), "Use vertical right element"
    Textfield (212,465 100x20), "%d", text variable: _20_AUTO.recipe.st120.xUseVerLeft
        OnMouseDown: write the text variable via Default
    Textfield (212,495 100x20), "%d", text variable: _20_AUTO.recipe.st120.xUseVerRight
        OnMouseDown: write the text variable via Default
    Textfield (210,240 100x20), "%d", text variable: _20_AUTO.recipe.st120.FeederConfigRight.InFilterDelay
        OnMouseDown: write the text variable via Default
    Textfield (210,270 100x20), "%d", text variable: _20_AUTO.recipe.st120.FeederConfigRight.StartDelay
        OnMouseDown: write the text variable via Default
    Textfield (210,300 100x20), "%d", text variable: _20_AUTO.recipe.st120.FeederConfigRight.StopDelay
        OnMouseDown: write the text variable via Default
    Textfield (210,330 100x20), "%d", text variable: _20_AUTO.recipe.st120.FeederConfigRight.EmptyDelay
        OnMouseDown: write the text variable via Default
    Label (100,55 200x20), "FeederConfig Left"
    Label (100,215 200x20), "FeederConfig Right"
    Label (1,240 200x20), "InFilterDelay"
    Label (1,270 200x20), "StartDelay"
    Label (1,300 200x20), "StopDelay"
    Label (1,330 200x20), "EmptyDelay"
    Label (2,385 200x20), "TON sensor tube presence left"
    Label (2,415 200x20), "TON sensor tube presence right"
    Textfield (212,385 100x20), "%d", text variable: _20_AUTO.recipe.st120.TON_PieceInSeperatorLeft
        OnMouseDown: write the text variable via Default
    Textfield (212,415 100x20), "%d", text variable: _20_AUTO.recipe.st120.TON_PieceInSeperatorRight
        OnMouseDown: write the text variable via Default
END_VISUALIZATION

// ---- POUs/20_AUTO/ST120/VISU_ST120.TcVIS
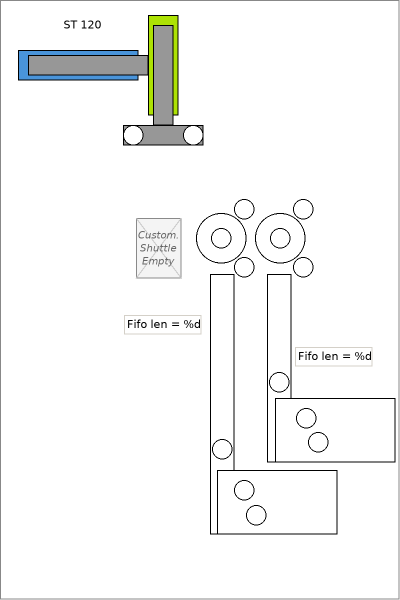
VISUALIZATION VISU_ST120  // 400x600
    Ellipse (196,213 50x50), colour toggle: GVL.st120_aut.fb_Feeder.fb_pivotLeft.xOUT_VALVE
    Image (136,218 45x60), invisible if: NOT __ISVALIDREF(GVL.st120_aut._Mover), image: Custom.Shuttle Empty
    Rectangle (18,50 120x30)
    Rectangle (28,55 120x20)
        p3560616238: GVL.st120_aut.fb_Pnp.fb_simu_axis120_01Y.rOUT_PixActual
    Rectangle (148,15 30x100)
        p3560616238: GVL.st120_aut.fb_Pnp.fb_simu_axis120_01Y.rOUT_PixActual
    Rectangle (153,25 20x100)
        p2738717112: GVL.st120_aut.fb_Pnp.fb_simu_axis120_02Z.rOUT_PixActual
        p3560616238: GVL.st120_aut.fb_Pnp.fb_simu_axis120_01Y.rOUT_PixActual
    Rectangle (210,274 24x260)
    Ellipse (212,439 20x20), colour toggle: GVL.st120_aut.fb_Feeder.simu_fifoLeft.IsFull()
    Ellipse (211,228 20x20), colour toggle: GVL.st120_aut.fb_Feeder.simu_fifoLeft.IsFull()
    Textfield (124,315 77x19), "Fifo len = %d", text variable: GVL.st120_aut.fb_Feeder.simu_fifoLeft.GetLen()
    Label (40,15 85x20), "ST 120"
    RoundedRectangle (217,470 120x64), colour toggle: GVL.st120_aut.fb_Feeder.fb_feederLeft.xOUT_EnableFeeder
    Rectangle (267,274 24x188)
    Ellipse (269,372 20x20), colour toggle: GVL.st120_aut.fb_Feeder.simu_fifoRight.IsFull()
    RoundedRectangle (275,398 120x64), colour toggle: GVL.st120_aut.fb_Feeder.fb_feederRight.xOUT_EnableFeeder
    Rectangle (123,125 80x20)
        p2738717112: GVL.st120_aut.fb_Pnp.fb_simu_axis120_02Z.rOUT_PixActual
        p3560616238: GVL.st120_aut.fb_Pnp.fb_simu_axis120_01Y.rOUT_PixActual
    Ellipse (183,125 20x20), colour toggle: GVL.st120_aut.fb_Pnp.fb_gripperRight.xIN_AS
        p3560616238: GVL.st120_aut.fb_Pnp.fb_simu_axis120_01Y.rOUT_PixActual
        p2738717112: GVL.st120_aut.fb_Pnp.fb_simu_axis120_02Z.rOUT_PixActual
    Ellipse (123,125 20x20), colour toggle: GVL.st120_aut.fb_Pnp.fb_gripperLeft.xIN_AS
        p3560616238: GVL.st120_aut.fb_Pnp.fb_simu_axis120_01Y.rOUT_PixActual
        p2738717112: GVL.st120_aut.fb_Pnp.fb_simu_axis120_02Z.rOUT_PixActual
    Textfield (295,347 77x19), "Fifo len = %d", text variable: GVL.st120_aut.fb_Feeder.simu_fifoRight.GetLen()
    Ellipse (255,213 50x50), colour toggle: GVL.st120_aut.fb_Feeder.fb_pivotRight.xOUT_VALVE
    Ellipse (270,228 20x20), colour toggle: GVL.st120_aut.fb_Feeder.simu_fifoRight.IsFull()
    Ellipse (293,199 20x20), colour toggle: GVL.st120_aut.fb_Feeder.fb_pivotRight.xIN_GS
    Ellipse (293,257 20x20), colour toggle: GVL.st120_aut.fb_Feeder.fb_pivotRight.xIN_AS
    Ellipse (234,199 20x20), colour toggle: GVL.st120_aut.fb_Feeder.fb_pivotLeft.xIN_GS
    Ellipse (234,257 20x20), colour toggle: GVL.st120_aut.fb_Feeder.fb_pivotLeft.xIN_AS
    Ellipse (246,505 20x20), colour toggle: GVL.st120_aut.fb_Feeder.fb_hubladerLeft.xIN_GS
    Ellipse (234,480 20x20), colour toggle: GVL.st120_aut.fb_Feeder.fb_hubladerLeft.xIN_AS
    Ellipse (296,408 20x20), colour toggle: GVL.st120_aut.fb_Feeder.fb_hubladerRight.xIN_AS
    Ellipse (308,432 20x20), colour toggle: GVL.st120_aut.fb_Feeder.fb_hubladerRight.xIN_GS
END_VISUALIZATION

// ---- POUs/20_AUTO/ST125/VISU_Recipe_ST125.TcVIS
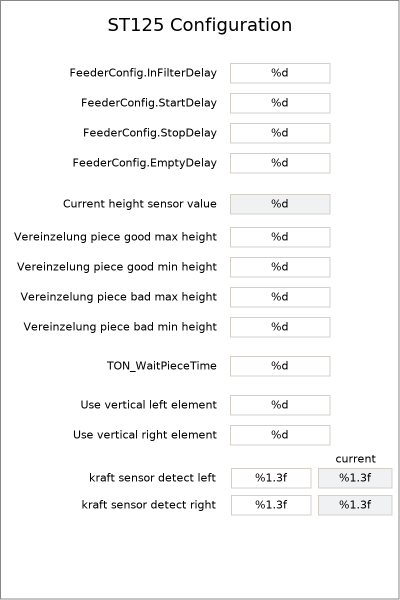
VISUALIZATION VISU_Recipe_ST125  // 400x600
    Textfield (230,63 100x20), "%d", text variable: _20_AUTO.recipe.st125.FeederConfig.InFilterDelay
        OnMouseDown: write the text variable via Default
    Label (0,5 400x40), "ST125 Configuration"
    Label (20,63 200x20), "FeederConfig.InFilterDelay"
    Textfield (230,93 100x20), "%d", text variable: _20_AUTO.recipe.st125.FeederConfig.StartDelay
        OnMouseDown: write the text variable via Default
    Label (20,93 200x20), "FeederConfig.StartDelay"
    Textfield (230,123 100x20), "%d", text variable: _20_AUTO.recipe.st125.FeederConfig.StopDelay
        OnMouseDown: write the text variable via Default
    Label (20,123 200x20), "FeederConfig.StopDelay"
    Textfield (230,153 100x20), "%d", text variable: _20_AUTO.recipe.st125.FeederConfig.EmptyDelay
        OnMouseDown: write the text variable via Default
    Label (20,153 200x20), "FeederConfig.EmptyDelay"
    Label (20,395 200x20), "Use vertical left element"
    Label (20,425 200x20), "Use vertical right element"
    Textfield (230,395 100x20), "%d", text variable: _20_AUTO.recipe.st125.xUseVerLeft
        OnMouseDown: write the text variable via Default
    Textfield (230,425 100x20), "%d", text variable: _20_AUTO.recipe.st125.xUseVerRight
        OnMouseDown: write the text variable via Default
    Textfield (230,227 100x20), "%d", text variable: _20_AUTO.recipe.st125.diPieceGoodMaxHeight
        OnMouseDown: write the text variable via Default
    Label (20,227 200x20), "Vereinzelung piece good max height"
    Textfield (230,257 100x20), "%d", text variable: _20_AUTO.recipe.st125.diPieceGoodMinHeight
        OnMouseDown: write the text variable via Default
    Label (20,257 200x20), "Vereinzelung piece good min height"
    Textfield (230,287 100x20), "%d", text variable: _20_AUTO.recipe.st125.diPieceWrongMaxHeight
        OnMouseDown: write the text variable via Default
    Label (20,287 200x20), "Vereinzelung piece bad max height"
    Textfield (230,317 100x20), "%d", text variable: _20_AUTO.recipe.st125.diPieceWrongMinHeight
        OnMouseDown: write the text variable via Default
    Label (20,317 200x20), "Vereinzelung piece bad min height"
    Textfield (230,194 100x20), "%d", text variable: IN.AI21_ST125_piece_height
    Label (20,194 200x20), "Current height sensor value"
    Textfield (230,356 100x20), "%d", text variable: _20_AUTO.recipe.st125.TON_WaitPieceTime
        OnMouseDown: write the text variable via Default
    Label (20,356 200x20), "TON_WaitPieceTime"
    Label (19,495 200x20), "kraft sensor detect right"
    Textfield (231,495 80x20), "%1.3f", text variable: _20_AUTO.recipe.st125.kraft_right_raw
        OnMouseDown: write the text variable via Default
    Label (19,468 200x20), "kraft sensor detect left"
    Textfield (231,468 80x20), "%1.3f", text variable: _20_AUTO.recipe.st125.kraft_left_raw
        OnMouseDown: write the text variable via Default
    Textfield (318,468 74x20), "%1.3f", text variable: GVL.st125_aut.fb_Pnp.fb_kraftLeft.lrOUT_value
        OnMouseDown: write the text variable via Default
    Textfield (318,495 74x20), "%1.3f", text variable: GVL.st125_aut.fb_Pnp.fb_kraftRight.lrOUT_value
        OnMouseDown: write the text variable via Default
    Label (321,449 70x20), "current"
END_VISUALIZATION

// ---- POUs/20_AUTO/ST125/VISU_ST125.TcVIS
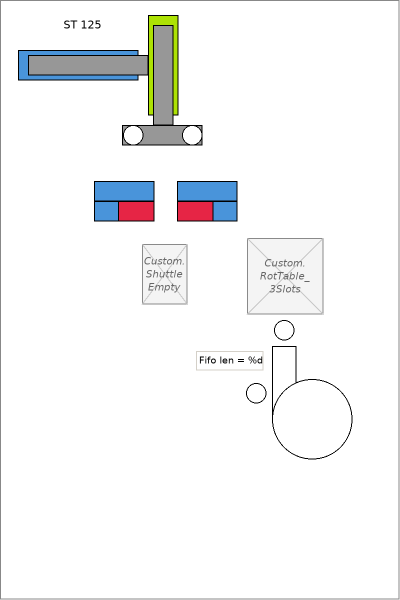
VISUALIZATION VISU_ST125  // 400x600
    Rectangle (187,201 50x20), invisible if: GVL.st125_aut.fb_Pnp.fb_handlingSolerohrRight.xIN_GS
    Rectangle (94,201 50x20), invisible if: GVL.st125_aut.fb_Pnp.fb_handlingSolerohrLeft.xIN_GS
    Rectangle (94,181 60x20), invisible if: GVL.st125_aut.fb_Pnp.fb_handlingSolerohrLeft.xIN_AS
    Rectangle (177,181 60x20), invisible if: GVL.st125_aut.fb_Pnp.fb_handlingSolerohrRight.xIN_AS
    Image (142,244 45x60), invisible if: NOT __ISVALIDREF(GVL.st125_aut._Mover), image: Custom.Shuttle Empty
    Image (247,238 76x76), image: Custom.RotTable_3Slots
        p2858320360: ST125_Axis.axis125_10W.rActPos
    Rectangle (18,50 120x30)
    Rectangle (28,55 120x20)
        p3560616238: GVL.st125_aut.fb_Pnp.fb_simu_axis125_01Y.rOUT_PixActual
    Rectangle (148,15 30x100)
        p3560616238: GVL.st125_aut.fb_Pnp.fb_simu_axis125_01Y.rOUT_PixActual
    Rectangle (153,25 20x100)
        p2738717112: GVL.st125_aut.fb_Pnp.fb_simu_axis125_02Z.rOUT_PixActual
        p3560616238: GVL.st125_aut.fb_Pnp.fb_simu_axis125_01Y.rOUT_PixActual
    Rectangle (272,346 24x73)
    Ellipse (272,379 80x80), colour toggle: GVL.st125_aut.fb_Feeder.simu_feeder.xIN_Enable
    Ellipse (246,383 20x20), colour toggle: GVL.st125_aut.fb_Feeder.simu_feeder.xOUT_NewPiece
    Ellipse (274,320 20x20)
    Textfield (196,351 67x19), "Fifo len = %d", text variable: GVL.st125_aut.fb_Feeder.simu_fifo_feeder_to_rotTable.GetLen()
    Label (40,15 85x20), "ST 125"
    Rectangle (122,125 80x20)
        p2738717112: GVL.st125_aut.fb_Pnp.fb_simu_axis125_02Z.rOUT_PixActual
        p3560616238: GVL.st125_aut.fb_Pnp.fb_simu_axis125_01Y.rOUT_PixActual
    Ellipse (123,125 20x20), colour toggle: GVL.st125_aut.fb_Pnp.fb_gripperFilterhutLeft.xIN_AS
        p3560616238: GVL.st125_aut.fb_Pnp.fb_simu_axis125_01Y.rOUT_PixActual
        p2738717112: GVL.st125_aut.fb_Pnp.fb_simu_axis125_02Z.rOUT_PixActual
    Ellipse (182,125 20x20), colour toggle: GVL.st125_aut.fb_Pnp.fb_gripperFilterhutRight.xIN_AS
        p3560616238: GVL.st125_aut.fb_Pnp.fb_simu_axis125_01Y.rOUT_PixActual
        p2738717112: GVL.st125_aut.fb_Pnp.fb_simu_axis125_02Z.rOUT_PixActual
    Rectangle (118,201 36x20), invisible if: NOT GVL.st125_aut.fb_Pnp.fb_gripperSolerohrLeft.xIN_AS
    Rectangle (177,201 36x20), invisible if: NOT GVL.st125_aut.fb_Pnp.fb_gripperSolerohrRight.xIN_AS
END_VISUALIZATION

// ---- POUs/20_AUTO/ST128/VISU_ST128.TcVIS
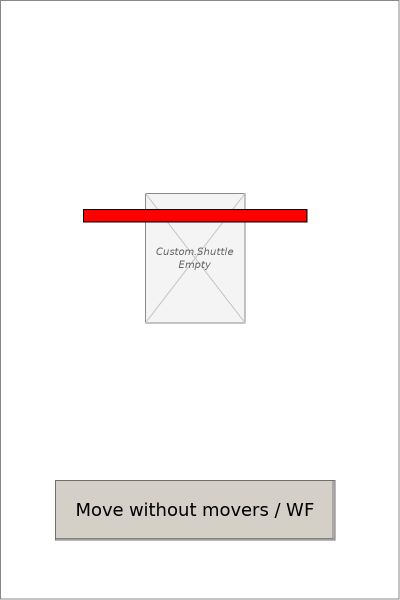
VISUALIZATION VISU_ST128  // 400x600
    Image (145,193 100x130), invisible if: NOT __ISVALIDREF(GVL.st128_aut._Mover), image: Custom.Shuttle Empty
        p2738717112: GVL.st128_aut.fb_TubeCapCheck.visu_shuttle_x_position
    Button (55,480 280x60), "Move without movers / WF", colour toggle: HMI.bArForceCyclusState[StationList_e.ST128]
        tap HMI.btArForceCyclus[StationList_e.ST128].button
    Rectangle (83,209 224x13)
END_VISUALIZATION

// ---- POUs/20_AUTO/ST130/VISU_Recipe_ST130.TcVIS
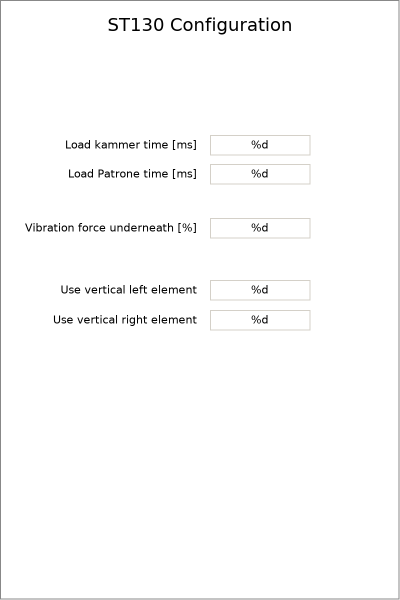
VISUALIZATION VISU_Recipe_ST130  // 400x600
    Label (0,5 400x40), "ST130 Configuration"
    Label (0,280 200x20), "Use vertical left element"
    Label (0,310 200x20), "Use vertical right element"
    Textfield (210,280 100x20), "%d", text variable: _20_AUTO.recipe.st130.xUseVerLeft
        OnMouseDown: write the text variable via Default
    Textfield (210,310 100x20), "%d", text variable: _20_AUTO.recipe.st130.xUseVerRight
        OnMouseDown: write the text variable via Default
    Label (0,135 200x20), "Load kammer time [ms]"
    Textfield (210,135 100x20), "%d", text variable: _20_AUTO.recipe.st130.diLoadKammer_ms
        OnMouseDown: write the text variable via Default
    Label (0,164 200x20), "Load Patrone time [ms]"
    Textfield (210,164 100x20), "%d", text variable: _20_AUTO.recipe.st130.diLoadPatrone_ms
        OnMouseDown: write the text variable via Default
    Label (0,218 200x20), "Vibration force underneath [%]"
    Textfield (210,218 100x20), "%d", text variable: _20_AUTO.recipe.st130.uiVibroUnderneath
        OnMouseDown: write the text variable via Default
END_VISUALIZATION

// ---- POUs/20_AUTO/ST130/VISU_ST130.TcVIS
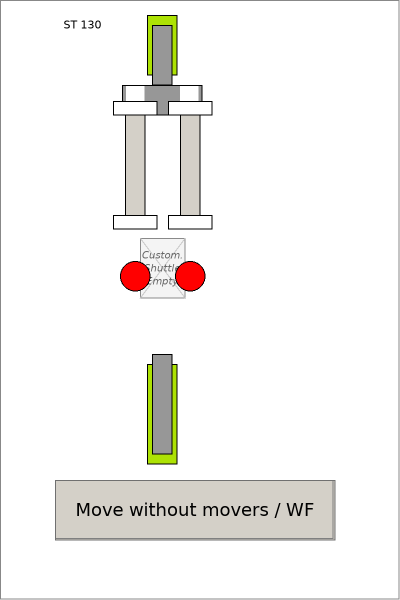
VISUALIZATION VISU_ST130  // 400x600
    RoundedRectangle (125,109 20x120)
    RoundedRectangle (180,109 20x120)
    Rectangle (106,7 116x108)
        p2738717112: GVL.st130_aut.fb_Dose.fb_simu_axis130_01Z.rOUT_PixActual
    Image (140,238 45x60), angle 90, invisible if: NOT __ISVALIDREF(GVL.st130_aut._Mover), image: Custom.Shuttle Empty
    Rectangle (147,15 30x60)
    Rectangle (152,25 20x60)
        p2738717112: GVL.st130_aut.fb_Dose.fb_simu_axis130_01Z.rOUT_PixActual
    Label (40,15 85x20), "ST 130"
    Rectangle (122,85 80x30)
        p2738717112: GVL.st130_aut.fb_Dose.fb_simu_axis130_01Z.rOUT_PixActual
    Rectangle (147,364 30x100)
    Rectangle (152,354 20x100)
        p2738717112: -GVL.st130_aut.fb_Dose.fb_simu_axis130_10Z.rOUT_PixActual
    Button (55,480 280x60), "Move without movers / WF", colour toggle: HMI.bArForceCyclusState[StationList_e.ST130]
        tap HMI.btArForceCyclus[StationList_e.ST130].button
    Rectangle (113,215 44x14), invisible if: NOT GVL.st130_aut.fb_Dose.fb_Kammer_Offnen_Rechts.xIN_GS
    Rectangle (168,215 44x14), invisible if: NOT GVL.st130_aut.fb_Dose.fb_Kammer_Offnen_Rechts.xIN_GS
    Rectangle (180,86 18x28)
        p2738717112: GVL.st130_aut.fb_Dose.fb_simu_axis130_01Z.rOUT_PixActual
    Rectangle (126,86 18x28)
        p2738717112: GVL.st130_aut.fb_Dose.fb_simu_axis130_01Z.rOUT_PixActual
    Rectangle (113,101 44x14), invisible if: NOT GVL.st130_aut.fb_Dose.fb_Kammer_nachfullen_Links.xIN_GS
        p2738717112: GVL.st130_aut.fb_Dose.fb_simu_axis130_01Z.rOUT_PixActual
    Rectangle (168,101 44x14), invisible if: NOT GVL.st130_aut.fb_Dose.fb_Kammer_nachfullen_Rechts.xIN_GS
        p2738717112: GVL.st130_aut.fb_Dose.fb_simu_axis130_01Z.rOUT_PixActual
    Ellipse (120,261 30x30), invisible if: NOT GVL.st130_aut.fb_Dose.fb_Niederhalter_Patrone.xIN_AS
    Ellipse (175,261 30x30), invisible if: NOT GVL.st130_aut.fb_Dose.fb_Niederhalter_Patrone.xIN_AS
END_VISUALIZATION

// ---- POUs/20_AUTO/ST140/VISU_Recipe_ST140.TcVIS
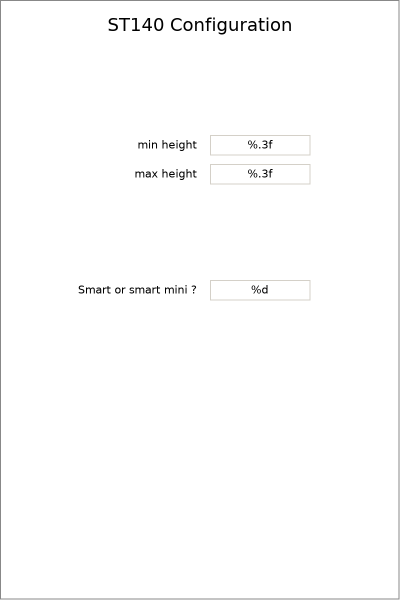
VISUALIZATION VISU_Recipe_ST140  // 400x600
    Label (0,5 400x40), "ST140 Configuration"
    Label (0,280 200x20), "Smart or smart mini ?"
    Textfield (210,280 100x20), "%d", text variable: _20_AUTO.recipe.st140.xIsTypeMiniOrSmart
        OnMouseDown: write the text variable via Default
    Label (0,135 200x20), "min height"
    Textfield (210,135 100x20), "%.3f", text variable: _20_AUTO.recipe.st140.rMinHeightSensor
        OnMouseDown: write the text variable via Default
    Label (0,164 200x20), "max height"
    Textfield (210,164 100x20), "%.3f", text variable: _20_AUTO.recipe.st140.rMaxHeightSensor
        OnMouseDown: write the text variable via Default
END_VISUALIZATION

// ---- POUs/20_AUTO/ST140/VISU_ST140.TcVIS
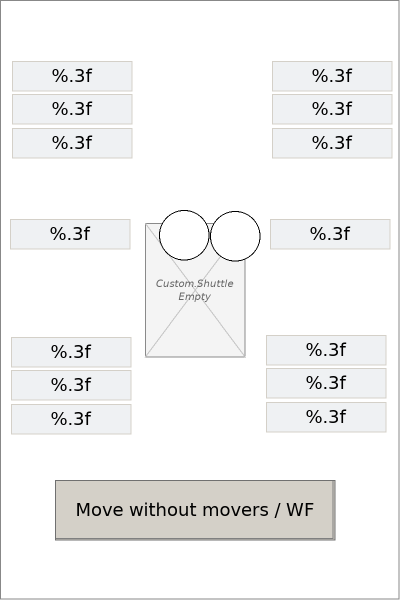
VISUALIZATION VISU_ST140  // 400x600
    Image (145,223 100x134), invisible if: NOT __ISVALIDREF(GVL.st140_aut._Mover), image: Custom.Shuttle Empty
        p3560616238: GVL.st140_aut.fb_Measure.visu_shuttle_x_position
    Button (55,480 280x60), "Move without movers / WF", colour toggle: HMI.bArForceCyclusState[StationList_e.ST140]
        tap HMI.btArForceCyclus[StationList_e.ST140].button
    Ellipse (159,210 50x50)
    Ellipse (210,211 50x50)
    Textfield (12,94 120x30), "%.3f", text variable: GVL.st140_aut.fb_Measure.arr_rMeasureTrack_Right[0][1]
    Textfield (12,128 120x30), "%.3f", text variable: GVL.st140_aut.fb_Measure.arr_rMeasureTrack_Right[0][2]
    Textfield (12,61 120x30), "%.3f", text variable: GVL.st140_aut.fb_Measure.arr_rMeasureTrack_Right[0][0]
    Textfield (272,94 120x30), "%.3f", text variable: GVL.st140_aut.fb_Measure.arr_rMeasureTrack_Right[1][1]
    Textfield (272,128 120x30), "%.3f", text variable: GVL.st140_aut.fb_Measure.arr_rMeasureTrack_Right[1][2]
    Textfield (272,61 120x30), "%.3f", text variable: GVL.st140_aut.fb_Measure.arr_rMeasureTrack_Right[1][0]
    Textfield (11,370 120x30), "%.3f", text variable: GVL.st140_aut.fb_Measure.arr_rMeasureTrack_Left[0][1]
    Textfield (11,404 120x30), "%.3f", text variable: GVL.st140_aut.fb_Measure.arr_rMeasureTrack_Left[0][2]
    Textfield (11,337 120x30), "%.3f", text variable: GVL.st140_aut.fb_Measure.arr_rMeasureTrack_Left[0][0]
    Textfield (266,368 120x30), "%.3f", text variable: GVL.st140_aut.fb_Measure.arr_rMeasureTrack_Left[1][1]
    Textfield (266,402 120x30), "%.3f", text variable: GVL.st140_aut.fb_Measure.arr_rMeasureTrack_Left[1][2]
    Textfield (266,335 120x30), "%.3f", text variable: GVL.st140_aut.fb_Measure.arr_rMeasureTrack_Left[1][0]
    Textfield (10,219 120x30), "%.3f", text variable: TO_REAL(IN.AI01_ST140_level_track_side)/1000.0
    Textfield (270,219 120x30), "%.3f", text variable: TO_REAL(IN.AI02_ST140_level_door_side)/1000.0
END_VISUALIZATION

// ---- POUs/20_AUTO/ST145/VISU_Recipe_ST145.TcVIS
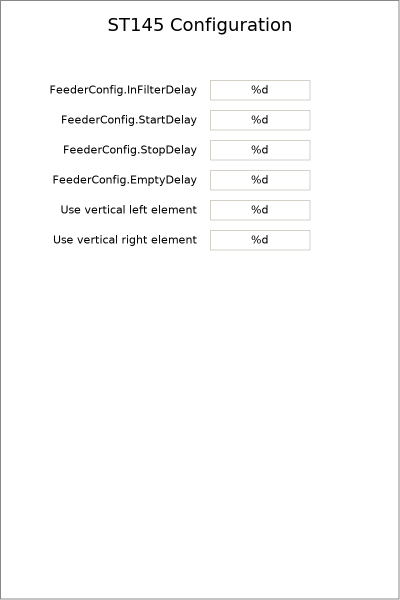
VISUALIZATION VISU_Recipe_ST145  // 400x600
    Textfield (210,80 100x20), "%d", text variable: _20_AUTO.recipe.st145.FeederConfig.InFilterDelay
        OnMouseDown: write the text variable via Default
    Label (0,5 400x40), "ST145 Configuration"
    Label (0,80 200x20), "FeederConfig.InFilterDelay"
    Textfield (210,110 100x20), "%d", text variable: _20_AUTO.recipe.st145.FeederConfig.StartDelay
        OnMouseDown: write the text variable via Default
    Label (0,110 200x20), "FeederConfig.StartDelay"
    Textfield (210,140 100x20), "%d", text variable: _20_AUTO.recipe.st145.FeederConfig.StopDelay
        OnMouseDown: write the text variable via Default
    Label (0,140 200x20), "FeederConfig.StopDelay"
    Textfield (210,170 100x20), "%d", text variable: _20_AUTO.recipe.st145.FeederConfig.EmptyDelay
        OnMouseDown: write the text variable via Default
    Label (0,170 200x20), "FeederConfig.EmptyDelay"
    Label (0,200 200x20), "Use vertical left element"
    Label (0,230 200x20), "Use vertical right element"
    Textfield (210,200 100x20), "%d", text variable: _20_AUTO.recipe.st145.xUseVerLeft
        OnMouseDown: write the text variable via Default
    Textfield (210,230 100x20), "%d", text variable: _20_AUTO.recipe.st145.xUseVerRight
        OnMouseDown: write the text variable via Default
END_VISUALIZATION

// ---- POUs/20_AUTO/ST145/VISU_ST145.TcVIS
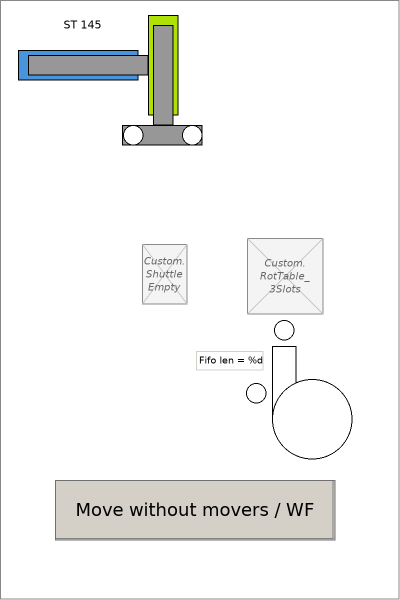
VISUALIZATION VISU_ST145  // 400x600
    Image (142,244 45x60), invisible if: NOT __ISVALIDREF(GVL.st145_aut._Mover), image: Custom.Shuttle Empty
    Image (247,238 76x76), image: Custom.RotTable_3Slots
        p2858320360: ST145_Axis.axis145_10W.rActPos
    Rectangle (18,50 120x30)
    Rectangle (28,55 120x20)
        p3560616238: GVL.st145_aut.fb_Pnp.fb_simu_axis145_01Y.rOUT_PixActual
    Rectangle (148,15 30x100)
        p3560616238: GVL.st145_aut.fb_Pnp.fb_simu_axis145_01Y.rOUT_PixActual
    Rectangle (153,25 20x100)
        p2738717112: GVL.st145_aut.fb_Pnp.fb_simu_axis145_02Z.rOUT_PixActual
        p3560616238: GVL.st145_aut.fb_Pnp.fb_simu_axis145_01Y.rOUT_PixActual
    Rectangle (272,346 24x73)
    Ellipse (272,379 80x80), colour toggle: GVL.st145_aut.fb_Feeder.simu_feeder.xIN_Enable
    Ellipse (246,383 20x20), colour toggle: GVL.st145_aut.fb_Feeder.simu_feeder.xOUT_NewPiece
    Ellipse (274,320 20x20), colour toggle: NOT GVL.st145_aut.fb_Feeder.simu_fifo_feeder_to_rotTable.IsEmpty()
    Textfield (196,351 67x19), "Fifo len = %d", text variable: GVL.st145_aut.fb_Feeder.simu_fifo_feeder_to_rotTable.GetLen()
    Label (40,15 85x20), "ST 145"
    Rectangle (122,125 80x20)
        p2738717112: GVL.st145_aut.fb_Pnp.fb_simu_axis145_02Z.rOUT_PixActual
        p3560616238: GVL.st145_aut.fb_Pnp.fb_simu_axis145_01Y.rOUT_PixActual
    Ellipse (123,125 20x20), colour toggle: GVL.st145_aut.fb_Pnp.fb_vakumGriperLeft.xIN_AS
        p3560616238: GVL.st145_aut.fb_Pnp.fb_simu_axis145_01Y.rOUT_PixActual
        p2738717112: GVL.st145_aut.fb_Pnp.fb_simu_axis145_02Z.rOUT_PixActual
    Ellipse (182,125 20x20), colour toggle: GVL.st145_aut.fb_Pnp.fb_vakumGriperRight.xIN_AS
        p3560616238: GVL.st145_aut.fb_Pnp.fb_simu_axis145_01Y.rOUT_PixActual
        p2738717112: GVL.st145_aut.fb_Pnp.fb_simu_axis145_02Z.rOUT_PixActual
    Button (55,480 280x60), "Move without movers / WF", colour toggle: HMI.bArForceCyclusState[StationList_e.ST145]
        tap HMI.btArForceCyclus[StationList_e.ST145].button
END_VISUALIZATION

// ---- POUs/20_AUTO/ST15x/VISU_Recipe_ST150.TcVIS
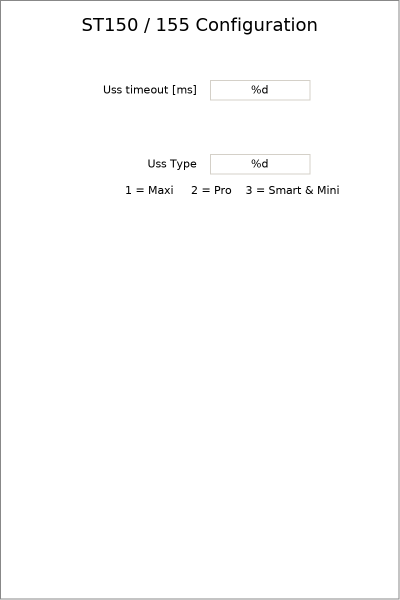
VISUALIZATION VISU_Recipe_ST150  // 400x600
    Textfield (210,80 100x20), "%d", text variable: _20_AUTO.recipe.st150.USS_ErrorTime_ms
        OnMouseDown: write the text variable via Default
    Label (0,5 400x40), "ST150 / 155 Configuration"
    Label (0,80 200x20), "Uss timeout [ms]"
    Textfield (210,154 100x20), "%d", text variable: _20_AUTO.recipe.st150.USS_Type
        OnMouseDown: write the text variable via Default
    Label (0,154 200x20), "Uss Type"
    Label (112,176 241x29), "1 = Maxi 2 = Pro 3 = Smart & Mini"
END_VISUALIZATION

// ---- POUs/20_AUTO/ST15x/VISU_ST150.TcVIS
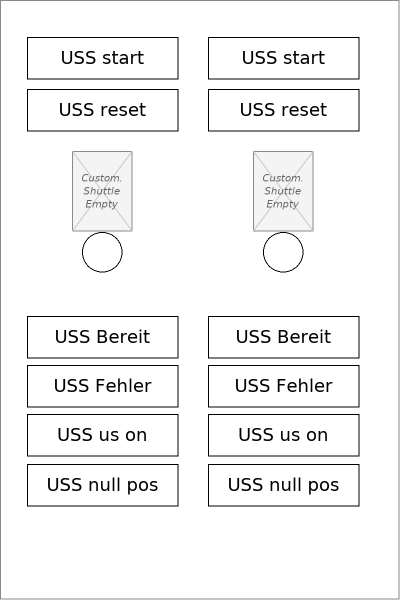
VISUALIZATION VISU_ST150  // 400x600
    RoundedRectangle (27,316 151x42), "USS Bereit", colour toggle: GVL.st150_aut.fb_Uss.xIN_welding_bits.Bereit
    RoundedRectangle (27,365 151x42), "USS Fehler", colour toggle: GVL.st150_aut.fb_Uss.xIN_welding_bits.Fehler
    RoundedRectangle (27,414 151x42), "USS us on", colour toggle: GVL.st150_aut.fb_Uss.xIN_welding_bits.US_on
    RoundedRectangle (27,464 151x42), "USS null pos", colour toggle: GVL.st150_aut.fb_Uss.xIN_welding_bits.NullPosition
    RoundedRectangle (27,37 151x42), "USS start", colour toggle: GVL.st150_aut.fb_Uss.xOUT_welding_bits.Start
    RoundedRectangle (27,89 151x42), "USS reset", colour toggle: GVL.st150_aut.fb_Uss.xOUT_welding_bits.Reset
    Ellipse (82,232 40x40), colour toggle: GVL.st150_aut.fb_Uss.xIN_capDetector
    Image (72,151 60x80), angle 90, invisible if: NOT __ISVALIDREF(GVL.st150_aut._Mover), image: Custom.Shuttle Empty
    RoundedRectangle (208,316 151x42), "USS Bereit", colour toggle: GVL.st155_aut.fb_Uss.xIN_welding_bits.Bereit
    RoundedRectangle (208,365 151x42), "USS Fehler", colour toggle: GVL.st155_aut.fb_Uss.xIN_welding_bits.Fehler
    RoundedRectangle (208,414 151x42), "USS us on", colour toggle: GVL.st155_aut.fb_Uss.xIN_welding_bits.US_on
    RoundedRectangle (208,464 151x42), "USS null pos", colour toggle: GVL.st155_aut.fb_Uss.xIN_welding_bits.NullPosition
    RoundedRectangle (208,37 151x42), "USS start", colour toggle: GVL.st155_aut.fb_Uss.xOUT_welding_bits.Start
    RoundedRectangle (208,89 151x42), "USS reset", colour toggle: GVL.st155_aut.fb_Uss.xOUT_welding_bits.Reset
    Ellipse (263,232 40x40), colour toggle: GVL.st155_aut.fb_Uss.xIN_capDetector
    Image (253,151 60x80), angle 90, invisible if: NOT __ISVALIDREF(GVL.st155_aut._Mover), image: Custom.Shuttle Empty
END_VISUALIZATION

// ---- POUs/20_AUTO/ST16x/VISU_Recipe_ST160.TcVIS
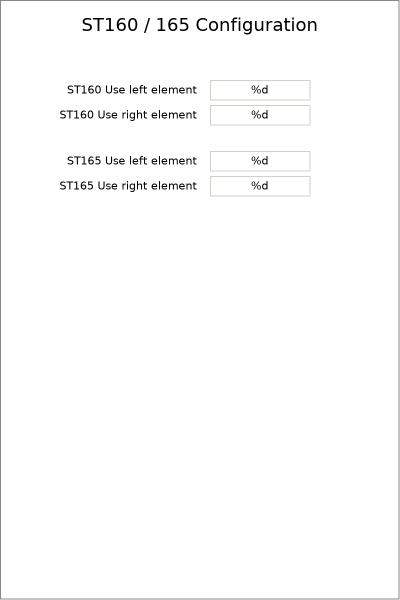
VISUALIZATION VISU_Recipe_ST160  // 400x600
    Textfield (210,80 100x20), "%d", text variable: _20_AUTO.recipe.st160.Use_element_left
        OnMouseDown: write the text variable via Default
    Label (0,5 400x40), "ST160 / 165 Configuration"
    Label (0,80 200x20), "ST160 Use left element"
    Textfield (210,105 100x20), "%d", text variable: _20_AUTO.recipe.st160.Use_element_right
        OnMouseDown: write the text variable via Default
    Label (0,105 200x20), "ST160 Use right element"
    Textfield (210,151 100x20), "%d", text variable: _20_AUTO.recipe.st165.Use_element_left
        OnMouseDown: write the text variable via Default
    Label (0,151 200x20), "ST165 Use left element"
    Textfield (210,176 100x20), "%d", text variable: _20_AUTO.recipe.st165.Use_element_right
        OnMouseDown: write the text variable via Default
    Label (0,176 200x20), "ST165 Use right element"
END_VISUALIZATION

// ---- POUs/20_AUTO/ST16x/VISU_ST160.TcVIS
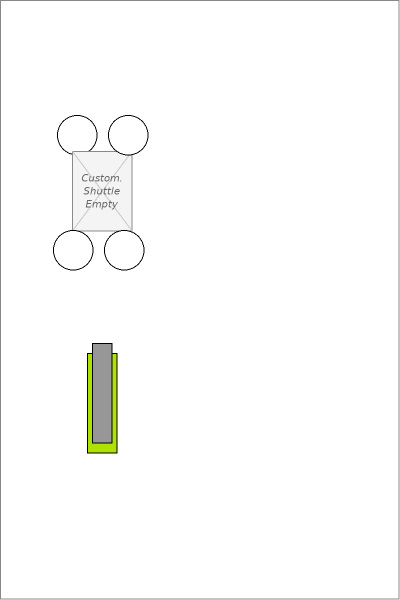
VISUALIZATION VISU_ST160  // 400x600
    Ellipse (57,115 40x40), colour toggle: GVL.st160_aut.fb_ABL_CETA.fb_capMainteningLeft.xIN_AS
    Image (72,151 60x80), angle 90, invisible if: NOT __ISVALIDREF(GVL.st160_aut._Mover), image: Custom.Shuttle Empty
    Ellipse (108,115 40x40), colour toggle: GVL.st160_aut.fb_ABL_CETA.fb_capMainteningRight.xIN_AS
    Rectangle (87,353 30x100)
    Rectangle (92,343 20x100)
        p2738717112: -GVL.st160_aut.fb_ABL_CETA.simu_axis160_01Z.rOUT_PixActual
    Ellipse (53,230 40x40), colour toggle: GVL.st160_aut.fb_ABL_CETA.fb_dichtung_left.xIN_AS
    Ellipse (104,230 40x40), colour toggle: GVL.st160_aut.fb_ABL_CETA.fb_dichtung_right.xIN_AS
END_VISUALIZATION

// ---- POUs/20_AUTO/ST170/VISU_Recipe_ST170.TcVIS
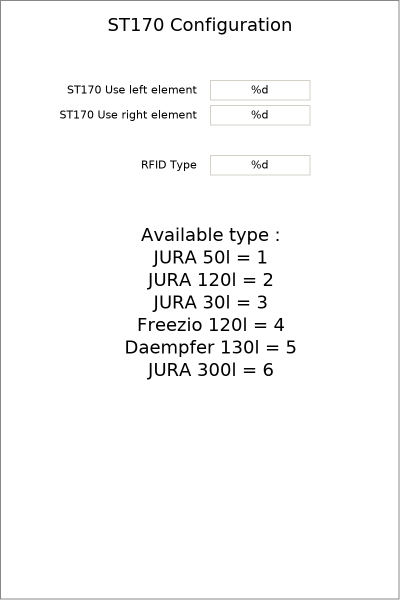
VISUALIZATION VISU_Recipe_ST170  // 400x600
    Textfield (210,80 100x20), "%d", text variable: _20_AUTO.recipe.st170.Use_element_left
        OnMouseDown: write the text variable via Default
    Label (0,5 400x40), "ST170 Configuration"
    Label (0,80 200x20), "ST170 Use left element"
    Textfield (210,105 100x20), "%d", text variable: _20_AUTO.recipe.st170.Use_element_right
        OnMouseDown: write the text variable via Default
    Label (0,105 200x20), "ST170 Use right element"
    Textfield (210,155 100x20), "%d", text variable: _20_AUTO.recipe.st170.RFID_Type
        OnMouseDown: write the text variable via Default
    Label (0,155 200x20), "RFID Type"
    Label (70,203 282x199), "Available type : JURA 50l = 1 JURA 120l = 2 JURA 30l = 3 Freezio 120l = 4 Daempfer 130l = 5 JURA 300l = 6"
END_VISUALIZATION

// ---- POUs/20_AUTO/ST170/VISU_ST170.TcVIS
